(* IEC 61131-3 sources: Yaha/Documentation/Infomaterial/OSCAT/pcworx_basic_333/module_export (part 2) *)

(* ---- CALIBRATE.ST ---- *)
(*@PROPERTIES_EX@
TYPE: POU
LOCALE: 0
IEC_LANGUAGE: ST
PLC_TYPE: independent
PROC_TYPE: independent
GROUP: ENGINEERING.MEASUREMENTS
*)
(*@KEY@:DESCRIPTION*)
version 1.3	11. mar. 2009
programmer 	hugo
tested BY	hans

Calibrate allows for offset and scale calibration of an analog input.
offset is calibrated to a stored reference Y_offset while CO is true.
after the offset is calibrated, scale can be calibrated to a reference value Y_scale while CS is true.
*)
(*@KEY@:END_DESCRIPTION*)
FUNCTION_BLOCK CALIBRATE

(*Group:Default*)

VAR_INPUT
	X :	REAL;
	CO :	BOOL;
	CS :	BOOL;
	Y_OFFSET :	REAL;
	Y_SCALE :	REAL;
END_VAR

VAR_OUTPUT
	Y :	REAL;
END_VAR

VAR RETAIN
	offset :	REAL;
	Scale :	REAL := 1.0;
END_VAR

(*@KEY@: WORKSHEET
NAME: CALIBRATE
IEC_LANGUAGE: ST
*)
(* check for calibration *)
IF CO THEN
	OFFSET := Y_Offset - X;
ELSIF CS THEN
	SCALE := Y_scale / (X + OFFSET);
END_IF;
(* calculate output *)
Y := (X + OFFSET) * SCALE;

(* revision history
hm 22.2.2007		rev 1.2
	changed VAR RETAIN PERSISTENT to VAR RETAIN for better compatibility
	wago lon contollers do not support persisitent

hm	11. mar. 2009	rev 1.3
	changed real constants to use dot syntax

*)
(*@KEY@: END_WORKSHEET *)
END_FUNCTION_BLOCK

(* ---- CAPITALIZE.ST ---- *)
(*@PROPERTIES_EX@
TYPE: POU
LOCALE: 0
IEC_LANGUAGE: ST
PLC_TYPE: independent
PROC_TYPE: independent
GROUP: STRINGS
*)
(*@KEY@:DESCRIPTION*)
version 1.1	29. mar 2008
programmer 	hugo
tested by	tobias

uppercase returns str while all letters a..z and ä,ö,ü are converted to uppercase
(*@KEY@:END_DESCRIPTION*)
FUNCTION_BLOCK CAPITALIZE

(*Group:Default*)

VAR_INPUT
	STR :	STRING;
END_VAR

VAR_OUTPUT
	CAPITALIZE :	STRING;
END_VAR

VAR
	char :	BYTE;
	char2 :	BYTE;
	pos :	INT;
	L :	INT;
	first :	BOOL;
	str_temp :	STRING;
END_VAR

(*@KEY@: WORKSHEET
NAME: CAPITALIZE
IEC_LANGUAGE: ST
*)
CAPITALIZE := str;
first := TRUE;
L := LEN(str);
FOR pos := 1 TO L DO
   	char := INT_TO_BYTE(GET_CHAR(str,pos));
	IF first THEN
		char2 := TO_UPPER(char);
    	IF char <> char2 THEN
    		str_temp := CAPITALIZE;
      		CAPITALIZE := REPLACE(str_temp,BYTE_TO_STRING(char2,'%c'),1,pos);
		END_IF;
	END_IF;
	(* remember in first if the next char needs to capitalized *)
	first := char = BYTE#32;
END_FOR;

(* revision histroy
hm		4. mar 2008	rev 1.0
	original release

hm	29. mar. 2008	rev 1.1
	changed STRING to STRING(STRING_LENGTH)
*)
(*@KEY@: END_WORKSHEET *)
END_FUNCTION_BLOCK

(* ---- CARG.ST ---- *)
(*@PROPERTIES_EX@
TYPE: POU
LOCALE: 0
IEC_LANGUAGE: ST
PLC_TYPE: independent
PROC_TYPE: independent
GROUP: MATHEMATICAL.COMPLEX
*)
(*@KEY@:DESCRIPTION*)
version 1.1	20. apr. 2008
programmer 	hugo
tested by	oscat

this function calculates the phase angle (argument) of a complex number
(*@KEY@:END_DESCRIPTION*)
FUNCTION_BLOCK CARG

(*Group:Default*)

VAR_INPUT
	X :	oscat_complex;
END_VAR

VAR_OUTPUT
	CARG :	REAL;
END_VAR

(*@KEY@: WORKSHEET
NAME: CARG
IEC_LANGUAGE: ST
*)
CARG := ATAN2(X.im, X.re);

(* revision history
hm	21. feb. 2008	rev 1.0
	original version

hm	20. apr. 2008	rev 1.1
	use ATAN2 instead of ATAN
*)
(*@KEY@: END_WORKSHEET *)
END_FUNCTION_BLOCK

(* ---- CASIN.ST ---- *)
(*@PROPERTIES_EX@
TYPE: POU
LOCALE: 0
IEC_LANGUAGE: ST
PLC_TYPE: independent
PROC_TYPE: independent
GROUP: MATHEMATICAL.COMPLEX
*)
(*@KEY@:DESCRIPTION*)
version 1.0	21 feb 2008
programmer 	hugo
tested by	oscat

this function calculates the arcus sinus function of a complex number
(*@KEY@:END_DESCRIPTION*)
FUNCTION_BLOCK CASIN

(*Group:Default*)

VAR_INPUT
	X :	oscat_complex;
END_VAR

VAR_OUTPUT
	CASIN :	oscat_complex;
END_VAR

VAR
	Y :	oscat_complex;
	CASINH :	CASINH;
END_VAR

(*@KEY@: WORKSHEET
NAME: CASIN
IEC_LANGUAGE: ST
*)
y.re := -x.im;
y.im := x.re;
CASINH(X:=y);
y := CASINH.CASINH;
CASIN.re := y.im;
CASIN.im := -y.re;

(* revision history
hm	21. feb 2008	rev 1.0
	original version

*)
(*@KEY@: END_WORKSHEET *)
END_FUNCTION_BLOCK

(* ---- CASINH.ST ---- *)
(*@PROPERTIES_EX@
TYPE: POU
LOCALE: 0
IEC_LANGUAGE: ST
PLC_TYPE: independent
PROC_TYPE: independent
GROUP: MATHEMATICAL.COMPLEX
*)
(*@KEY@:DESCRIPTION*)
version 1.0	21 feb 2008
programmer 	hugo
tested by	oscat

this function calculates the hyperbolic arcus sinus function of a complex number
(*@KEY@:END_DESCRIPTION*)
FUNCTION_BLOCK CASINH

(*Group:Default*)

VAR_INPUT
	X :	oscat_complex;
END_VAR

VAR_OUTPUT
	CASINH :	oscat_complex;
END_VAR

VAR
	Y :	oscat_complex;
	CLOG :	CLOG;
	CSQRT :	CSQRT;
END_VAR

(*@KEY@: WORKSHEET
NAME: CASINH
IEC_LANGUAGE: ST
*)
y.re := (X.re - X.im)*(X.re + X.im) + 1.0;
y.im := 2.0 * X.re * X.im;
CSQRT(X:=y);
y    := CSQRT.CSQRT;
y.re := y.re + x.re;
y.im := y.im + x.im;
CLOG(X:=y);
CASINH  := CLOG.CLOG;

(* revision history
hm	21. feb 2008	rev 1.0
	original version

*)
(*@KEY@: END_WORKSHEET *)
END_FUNCTION_BLOCK

(* ---- CATAN.ST ---- *)
(*@PROPERTIES_EX@
TYPE: POU
LOCALE: 0
IEC_LANGUAGE: ST
PLC_TYPE: independent
PROC_TYPE: independent
GROUP: MATHEMATICAL.COMPLEX
*)
(*@KEY@:DESCRIPTION*)
version 1.0	21 feb 2008
programmer 	hugo
tested by	oscat

this function calculates the complex arcus tangens
(*@KEY@:END_DESCRIPTION*)
FUNCTION_BLOCK CATAN

(*Group:Default*)

VAR_INPUT
	X :	oscat_complex;
END_VAR

VAR_OUTPUT
	CATAN :	oscat_complex;
END_VAR

VAR
	r2 :	REAL;
	num :	REAL;
	den :	REAL;
END_VAR

(*@KEY@: WORKSHEET
NAME: CATAN
IEC_LANGUAGE: ST
*)
r2 := x.re * x.re;
den := 1.0 - r2 - x.im * x.im;
CATAN.re := 0.5 * ATAN(2.0 * x.re / den);
num := x.im + 1.0;
num := r2 + num * num;
den := x.im - 1.0;
den := r2 + den * den;
CATAN.im := 0.25 * (LN(num)-LN(den));

(* revision history
hm	21. feb 2008	rev 1.0
	original version
*)
(*@KEY@: END_WORKSHEET *)
END_FUNCTION_BLOCK

(* ---- CATANH.ST ---- *)
(*@PROPERTIES_EX@
TYPE: POU
LOCALE: 0
IEC_LANGUAGE: ST
PLC_TYPE: independent
PROC_TYPE: independent
GROUP: MATHEMATICAL.COMPLEX
*)
(*@KEY@:DESCRIPTION*)
version 1.0	21 feb 2008
programmer 	hugo
tested by	oscat

this function calculates the complex arcus hyperbolic tangens
(*@KEY@:END_DESCRIPTION*)
FUNCTION_BLOCK CATANH

(*Group:Default*)

VAR_INPUT
	X :	oscat_complex;
END_VAR

VAR_OUTPUT
	CATANH :	oscat_complex;
END_VAR

VAR
	i2 :	REAL;
	num :	REAL;
	den :	REAL;
END_VAR

(*@KEY@: WORKSHEET
NAME: CATANH
IEC_LANGUAGE: ST
*)
i2 := x.im * x.im;
num := 1.0 + x.re;
num := i2 + num * num;
den := 1.0 - x.re;
den := i2 + den * den;
CATANH.re := 0.25 * (LN(num) - LN(den));
den := 1.0 - x.re * x.re - i2;
CATANH.im := 0.5 * ATAN(2.0 * x.im / den);

(* revision history
hm	21. feb 2008	rev 1.0
	original version

*)
(*@KEY@: END_WORKSHEET *)
END_FUNCTION_BLOCK

(* ---- CCON.ST ---- *)
(*@PROPERTIES_EX@
TYPE: POU
LOCALE: 0
IEC_LANGUAGE: ST
PLC_TYPE: independent
PROC_TYPE: independent
GROUP: MATHEMATICAL.COMPLEX
*)
(*@KEY@:DESCRIPTION*)
version 1.0	21 feb 2008
programmer 	hugo
tested by	oscat

this function calcucates the conjugation of a complex number
(*@KEY@:END_DESCRIPTION*)
FUNCTION_BLOCK CCON

(*Group:Default*)

VAR_INPUT
	X :	oscat_complex;
END_VAR

VAR_OUTPUT
	CCON :	oscat_complex;
END_VAR

(*@KEY@: WORKSHEET
NAME: CCON
IEC_LANGUAGE: ST
*)
CCON.re := x.re;
CCON.im := -x.im;

(* revision history
hm	21. feb 2008	rev 1.0
	original version

*)
(*@KEY@: END_WORKSHEET *)
END_FUNCTION_BLOCK

(* ---- CCOS.ST ---- *)
(*@PROPERTIES_EX@
TYPE: POU
LOCALE: 0
IEC_LANGUAGE: ST
PLC_TYPE: independent
PROC_TYPE: independent
GROUP: MATHEMATICAL.COMPLEX
*)
(*@KEY@:DESCRIPTION*)
version 1.0	21 feb 2008
programmer 	hugo
tested by	oscat

this function calculates the cosinus function of a complex number
(*@KEY@:END_DESCRIPTION*)
FUNCTION_BLOCK CCOS

(*Group:Default*)

VAR_INPUT
	X :	oscat_complex;
END_VAR

VAR_OUTPUT
	CCOS :	oscat_complex;
END_VAR

VAR
	CSET :	CSET;
	CCOSH :	CCOSH;
END_VAR

(*@KEY@: WORKSHEET
NAME: CCOS
IEC_LANGUAGE: ST
*)
CSET(RE:= -X.im,IM:=X.re);
CCOSH(X:=CSET.CSET);
CCOS := CCOSH.CCOSH;

(* revision history
hm	21. feb 2008	rev 1.0
	original version

*)
(*@KEY@: END_WORKSHEET *)
END_FUNCTION_BLOCK

(* ---- CCOSH.ST ---- *)
(*@PROPERTIES_EX@
TYPE: POU
LOCALE: 0
IEC_LANGUAGE: ST
PLC_TYPE: independent
PROC_TYPE: independent
GROUP: MATHEMATICAL.COMPLEX
*)
(*@KEY@:DESCRIPTION*)
version 1.0	21 feb 2008
programmer 	hugo
tested by	oscat

this function calculates the arcus tangens function of a complex number
(*@KEY@:END_DESCRIPTION*)
FUNCTION_BLOCK CCOSH

(*Group:Default*)

VAR_INPUT
	X :	oscat_complex;
END_VAR

VAR_OUTPUT
	CCOSH :	oscat_complex;
END_VAR

(*@KEY@: WORKSHEET
NAME: CCOSH
IEC_LANGUAGE: ST
*)
CCOSH.re := cosH(x.re) * COS(x.im);
CCOSH.im := sinH(x.re) * SIN(x.im);

(* revision history
hm	21. feb 2008	rev 1.0
	original version

*)
(*@KEY@: END_WORKSHEET *)
END_FUNCTION_BLOCK

(* ---- CDIV.ST ---- *)
(*@PROPERTIES_EX@
TYPE: POU
LOCALE: 0
IEC_LANGUAGE: ST
PLC_TYPE: independent
PROC_TYPE: independent
GROUP: MATHEMATICAL.COMPLEX
*)
(*@KEY@:DESCRIPTION*)
version 1.0	21 feb 2008
programmer 	hugo
tested by	oscat

this function divides two complex numbers
(*@KEY@:END_DESCRIPTION*)
FUNCTION_BLOCK CDIV

(*Group:Default*)

VAR_INPUT
	X :	oscat_complex;
	Y :	oscat_complex;
END_VAR

VAR_OUTPUT
	CDIV :	oscat_complex;
END_VAR

VAR
	temp :	REAL;
END_VAR

(*@KEY@: WORKSHEET
NAME: CDIV
IEC_LANGUAGE: ST
*)
temp := Y.re * Y.re + Y.im * Y.im;
IF temp = 0.0 THEN CDIV.re := 0.0;CDIV.im := 0.0;RETURN;END_IF;
CDIV.re := (X.re * Y.re + X.im * Y.im) / temp;
CDIV.im := (X.im * Y.re - X.re * Y.im) / temp;

(* revision history
hm	21. feb 2008	rev 1.0
	original version

*)
(*@KEY@: END_WORKSHEET *)
END_FUNCTION_BLOCK

(* ---- CEXP.ST ---- *)
(*@PROPERTIES_EX@
TYPE: POU
LOCALE: 0
IEC_LANGUAGE: ST
PLC_TYPE: independent
PROC_TYPE: independent
GROUP: MATHEMATICAL.COMPLEX
*)
(*@KEY@:DESCRIPTION*)
version 1.0	21 feb 2008
programmer 	hugo
tested by	oscat

this function calculates the complex exponent
(*@KEY@:END_DESCRIPTION*)
FUNCTION_BLOCK CEXP

(*Group:Default*)

VAR_INPUT
	X :	oscat_complex;
END_VAR

VAR_OUTPUT
	CEXP :	oscat_complex;
END_VAR

VAR
	Temp :	REAL;
END_VAR

(*@KEY@: WORKSHEET
NAME: CEXP
IEC_LANGUAGE: ST
*)
temp := EXP(X.re);
CEXP.re := temp * COS(X.im);
CEXP.im := temp * SIN(X.im);

(* revision history
hm	21. feb 2008	rev 1.0
	original version

*)
(*@KEY@: END_WORKSHEET *)
END_FUNCTION_BLOCK

(* ---- CHARCODE.ST ---- *)
(*@PROPERTIES_EX@
TYPE: POU
LOCALE: 0
IEC_LANGUAGE: ST
PLC_TYPE: independent
PROC_TYPE: independent
GROUP: STRINGS
*)
(*@KEY@:DESCRIPTION*)
version 1.1		19. oct. 2008
programmer 		hugo
tested by		hugo

CHARCODE converts a HTML Character NAME INTO ITS code
'äuml' is convterted to ä
'euro' is converted to €
(*@KEY@:END_DESCRIPTION*)
FUNCTION_BLOCK CHARCODE

(*Group:IN_OUT*)

VAR_INPUT
	STR :	oscat_STRING10;
END_VAR

VAR_OUTPUT
	CHARCODE :	BYTE;
END_VAR

VAR
	found :	oscat_STRING1;
	search :	oscat_STRING10;
	pos :	INT;
	CODE :	CODE;
	i :	INT;
	SETUP_CHARNAMES :	SETUP_CHARNAMES;
	CHARNAMES :	oscat_CHARNAMES;
END_VAR

(*@KEY@: WORKSHEET
NAME: CHARCODE
IEC_LANGUAGE: ST
*)
SETUP_CHARNAMES(CHARNAMES:=CHARNAMES);
CHARNAMES:=SETUP_CHARNAMES.CHARNAMES;

IF LEN(str) = 1 THEN
    CODE(STR:=STR,POS:=1);
    CHARCODE:=CODE.CODE;
ELSIF LEN(str) > 0 THEN
	(* construct search string *)
	search := CONCAT('&', str);
	search := CONCAT(search, ';');
	WHILE pos = 0 AND (i < 11) DO
		i := i + 1;
		pos := FIND(CHARNAMES[i], search);
	END_WHILE;
	found := MID(CHARNAMES[i], 1, pos - 1);
    CODE(STR:=found,POS:=1);
    CHARCODE:=CODE.CODE;
END_IF;

(* revision history
hm	13. may. 2008	rev 1.0
	original version

hm	19. oct. 2008	rev 1.1
	changed setup constants

hm	24. oct. 2008	rev 1.2
	optimized code
*)
(*@KEY@: END_WORKSHEET *)
END_FUNCTION_BLOCK

(* ---- CHARNAME.ST ---- *)
(*@PROPERTIES_EX@
TYPE: POU
LOCALE: 0
IEC_LANGUAGE: ST
PLC_TYPE: independent
PROC_TYPE: independent
GROUP: STRINGS
*)
(*@KEY@:DESCRIPTION*)
version 1.4		17. dec. 2008
programmer 		hugo
tested by		oscat

CHARNAME converts a Character code into its HTML character name
ä is convterted to 'äuml'
€ is converted to 'euro'
the character itself is returned if no name is available for the character
(*@KEY@:END_DESCRIPTION*)
FUNCTION_BLOCK CHARNAME

(*Group:IN_OUT*)

VAR_INPUT
	C :	BYTE;
END_VAR

VAR_OUTPUT
	CHARNAME :	oscat_STRING10;
END_VAR

VAR
	CHARNAME2 :	oscat_STRING10;
	pos :	INT;
	i :	INT;
	CHR_TO_STRING :	CHR_TO_STRING;
	SETUP_CHARNAMES :	SETUP_CHARNAMES;
	CHARNAMES :	oscat_CHARNAMES;
END_VAR

(*@KEY@: WORKSHEET
NAME: CHARNAME
IEC_LANGUAGE: ST
*)
SETUP_CHARNAMES(CHARNAMES:=CHARNAMES);
CHARNAMES:=SETUP_CHARNAMES.CHARNAMES;

IF C <> BYTE#0 THEN
	(* construct search string from code followed by $ sign, also clear charname string*)
	CHR_TO_STRING(C:=C);
	CHARNAME := CHR_TO_STRING.CHR_TO_STRING;
	CHARNAME2 := CONCAT(CHARNAME,'&');
	CHARNAME := CONCAT(';', CHARNAME2);
	WHILE pos = 0 AND (i < 11) DO
		i := i + 1;
		pos := FIND(CHARNAMES[i], CHARNAME);
	END_WHILE;
	IF pos > 0 THEN
		CHARNAME := MID(CHARNAMES[i], 10, pos + 3);
		(* search for end of name and truncate *)
		pos := FIND(CHARNAME, ';');
		CHARNAME := LEFT(CHARNAME,pos - 1);
	ELSE
		CHR_TO_STRING(C:=C);
		CHARNAME := CHR_TO_STRING.CHR_TO_STRING;
	END_IF;
ELSE
	CHARNAME := '';
END_IF;

(* revision history
hm	13. may. 2008	rev 1.0
	original version

hm	16. jun. 2008	rev 1.1
	changed nested call of concat for better compatibility

hm	19. oct. 2008	rev 1.2
	changes setup constants

hm	24. oct. 2008	rev 1.3
	new code for high performance

hm	17. dec. 2008	rev 1.4
	changed function chr to chr_to_string
*)
(*@KEY@: END_WORKSHEET *)
END_FUNCTION_BLOCK

(* ---- CHK_REAL.ST ---- *)
(*@PROPERTIES_EX@
TYPE: POU
LOCALE: 0
IEC_LANGUAGE: ST
PLC_TYPE: independent
PROC_TYPE: independent
GROUP: LOGIC.GATE_LOGIC
*)
(*@KEY@:DESCRIPTION*)
version 1.0	20. jan. 2011
programmer 	hugo
tested by	tobias

this function checks a floating point variable of type real (IEEE754-32Bits) for NAN and infinity
RETURN values: #0 = normal value, #20 = +infinity, #40 = -infinty, #80 = NAN

(*@KEY@:END_DESCRIPTION*)
FUNCTION_BLOCK CHK_REAL

(*Group:Default*)

VAR_INPUT
	X :	REAL;
END_VAR

VAR_OUTPUT
	CHK_REAL :	BYTE;
END_VAR

VAR
	tmp :	DWORD;
	REAL_TO_DW :	REAL_TO_DW;
END_VAR

(*@KEY@: WORKSHEET
NAME: CHK_REAL
IEC_LANGUAGE: ST
*)
REAL_TO_DW(X:=X); (* move real to dword, real_to_dword does not work becasze it treats dword as a number on many systems *)
tmp := ROL(REAL_TO_DW.REAL_TO_DW,1);(* rotate left foir easy checking, sign will be at lease significant digit *)
IF tmp < DWORD#16#FF000000 THEN
	CHK_REAL := BYTE#16#00;	(* normalized and denormalized numbers *)
ELSIF tmp = DWORD#16#FF000000 THEN
	CHK_REAL := BYTE#16#20;	(* X is +infinity see IEEE754 *)
ELSIF tmp = DWORD#16#FF000001 THEN
	CHK_REAL := BYTE#16#40;	(* X is -infinity see IEEE754 *)
ELSE
	CHK_REAL := BYTE#16#80;	(* X is NAN see IEEE754 *)
END_IF;

(* revision history
hm	 20. jan. 2011	rev 1.0
	original version

*)

(*@KEY@: END_WORKSHEET *)
END_FUNCTION_BLOCK

(* ---- CHR_TO_STRING.ST ---- *)
(*@PROPERTIES_EX@
TYPE: POU
LOCALE: 0
IEC_LANGUAGE: ST
PLC_TYPE: independent
PROC_TYPE: independent
GROUP: STRINGS
*)
(*@KEY@:DESCRIPTION*)
version 1.3	17. dec. 2008
programmer 	hugo
tested by	oscat

CHR creates a character from a byte input and stuffs it in a one character length string.
(*@KEY@:END_DESCRIPTION*)
FUNCTION_BLOCK CHR_TO_STRING

(*Group:x*)

VAR_INPUT
	C :	BYTE;
END_VAR

VAR_OUTPUT
	CHR_TO_STRING :	oscat_STRING1;
END_VAR

(*@KEY@: WORKSHEET
NAME: CHR_TO_STRING
IEC_LANGUAGE: ST
*)
CHR_TO_STRING := BYTE_TO_STRING(C,'%c');

(* revision history
hm	16 jan 2007		rev 1.0
	original version

hm	4. feb. 2008	rev 1.1
	return string would not be terminated properly

hm	29. mar. 2008	rev 1.2
	changed STRING to STRING(1)

hm	17. dec. 2008	rev 1.3
	changed name of function from chr to chr_to_string
*)
(*@KEY@: END_WORKSHEET *)
END_FUNCTION_BLOCK

(* ---- CINV.ST ---- *)
(*@PROPERTIES_EX@
TYPE: POU
LOCALE: 0
IEC_LANGUAGE: ST
PLC_TYPE: independent
PROC_TYPE: independent
GROUP: MATHEMATICAL.COMPLEX
*)
(*@KEY@:DESCRIPTION*)
version 1.0	21 feb 2008
programmer 	hugo
tested by	oscat

this function calculates the inverse of a complex numbers (1 / X)
(*@KEY@:END_DESCRIPTION*)
FUNCTION_BLOCK CINV

(*Group:Default*)

VAR_INPUT
	X :	oscat_complex;
END_VAR

VAR_OUTPUT
	CINV :	oscat_complex;
END_VAR

VAR
	temp :	REAL;
END_VAR

(*@KEY@: WORKSHEET
NAME: CINV
IEC_LANGUAGE: ST
*)
temp := X.re * X.re + X.im * X.im;
IF temp = 0.0 THEN CINV.re := 0.0;CINV.im := 0.0;RETURN;END_IF;
CINV.re := X.re / temp;
CINV.im := -X.im / temp;

(* revision history
hm	21. feb 2008	rev 1.0
	original version

*)
(*@KEY@: END_WORKSHEET *)
END_FUNCTION_BLOCK

(* ---- CLEAN.ST ---- *)
(*@PROPERTIES_EX@
TYPE: POU
LOCALE: 0
IEC_LANGUAGE: ST
PLC_TYPE: independent
PROC_TYPE: independent
GROUP: STRINGS
*)
(*@KEY@:DESCRIPTION*)
version 1.0	18. jun. 2008
programmer 	hugo
tested by	oscat

Clean deletes all characters from a string except the ones specified in CX.
(*@KEY@:END_DESCRIPTION*)
FUNCTION_BLOCK CLEAN

(*Group:lokal*)

(*Group:IN_OUT*)

VAR_INPUT
	IN :	oscat_STRING250;
	CX :	STRING;
END_VAR

VAR_OUTPUT
	CLEAN :	oscat_STRING250;
END_VAR

VAR
	pos :	INT;
	stop :	INT;
	char :	oscat_STRING1;
END_VAR

(*@KEY@: WORKSHEET
NAME: CLEAN
IEC_LANGUAGE: ST
*)
(* copy input string *)
CLEAN := IN;
stop := LEN(in);
pos := 1;
WHILE pos <= stop DO
    char := MID(CLEAN, 1, pos);
	IF FIND(cx,char) > 0 THEN
		(* charcter found skip to next one *)
		pos := pos + 1;
	ELSE
		(* wrong chracter needs to be deleted *)
		CLEAN := DELETE(CLEAN, 1, pos);
		stop := stop - 1;	(* the string is one character shorter now *)
	END_IF;
END_WHILE;

(* revision history

hm		18. jun. 2008	rev 1.0
	original version

*)
(*@KEY@: END_WORKSHEET *)
END_FUNCTION_BLOCK

(* ---- CLICK_CNT.ST ---- *)
(*@PROPERTIES_EX@
TYPE: POU
LOCALE: 0
IEC_LANGUAGE: ST
PLC_TYPE: independent
PROC_TYPE: independent
GROUP: LOGIC.GENERATORS
*)
(*@KEY@:DESCRIPTION*)
version 1.0	16. jul. 2008
programmer 	hugo
tested by	oscat

this Module decodes a specified number of clicks.
the output trig is high for one cycle if N clicks are present within a specified time TC.
(*@KEY@:END_DESCRIPTION*)
FUNCTION_BLOCK CLICK_CNT

(*Group:Default*)

VAR_INPUT
	IN :	BOOL;
	N :	INT;
	TC :	TIME;
END_VAR

VAR_OUTPUT
	Q :	BOOL;
END_VAR

VAR
	tx :	TP;
	edge :	BOOL;
	cnt :	INT := INT#-1;
END_VAR

(*@KEY@: WORKSHEET
NAME: CLICK_CNT
IEC_LANGUAGE: ST
*)
(* Q shall only be active for one cycle only *)
Q := FALSE;

IF in AND NOT edge AND NOT tx.q THEN
	(* a rising edge on in sets the counter to 0 *)
	cnt := 0;
ELSIF tx.Q AND NOT IN AND edge THEN
	(* count falling edges when tp.q is true *)
	cnt := cnt + 1;
ELSIF NOT tx.Q THEN
	Q := cnt=N;
	cnt := -1;
END_IF;

(* remember the status of IN *)
edge := IN;
tx(in := IN, pt := TC);

(* revision history

hm 	16. jul. 2008	rev 1.0
	original version released

*)
(*@KEY@: END_WORKSHEET *)
END_FUNCTION_BLOCK

(* ---- CLICK_DEC.ST ---- *)
(*@PROPERTIES_EX@
TYPE: POU
LOCALE: 0
IEC_LANGUAGE: ST
PLC_TYPE: independent
PROC_TYPE: independent
GROUP: LOGIC.GENERATORS
*)
(*@KEY@:DESCRIPTION*)
version 1.1	14. mar. 2009
programmer 	hugo
tested by	oscat

this Module detects a rising edge on In and decodes the amount of falling edges (Pulses) within a specified time TC.
the outputs Q0..Q3 will go true for one cycle and the amount of clicks within a specified time TC.
if only a rising egde is detected within TC Q0 will respond, Q1 for 1 pulse and so on..

(*@KEY@:END_DESCRIPTION*)
FUNCTION_BLOCK CLICK_DEC

(*Group:Default*)

VAR_INPUT
	IN :	BOOL;
	TC :	TIME;
END_VAR

VAR_OUTPUT
	Q0 :	BOOL;
	Q1 :	BOOL;
	Q2 :	BOOL;
	Q3 :	BOOL;
END_VAR

VAR
	tx :	TP;
	edge :	BOOL;
	cnt :	INT := INT#-1;
END_VAR

(*@KEY@: WORKSHEET
NAME: CLICK_DEC
IEC_LANGUAGE: ST
*)
(* Q shall only be active for one cycle only *)
IF in = FALSE THEN
	Q0 := FALSE;
	Q1 := FALSE;
	Q2 := FALSE;
	Q3 := FALSE;
END_IF;

IF in AND NOT edge AND NOT tx.q THEN
	(* a rising edge on in sets the counter to 0 *)
	cnt := 0;
ELSIF tx.Q AND NOT IN AND edge THEN
	(* count falling edges when tp.q is true *)
	cnt := cnt + 1;
ELSIF NOT tx.Q THEN
	CASE cnt OF
		0 : Q0 := TRUE;
		1 : Q1 := TRUE;
		2 : Q2 := TRUE;
		3 : Q3 := TRUE;
	END_CASE;
	cnt := -1;
END_IF;

(* remember the status of IN *)
edge := IN;
tx(in := IN, pt := TC);

(* revision history

hm 17. jul. 2008	rev 1.0
	original version released

hm	14. mar. 2009	rev 1.1
	removed double assignments

*)
(*@KEY@: END_WORKSHEET *)
END_FUNCTION_BLOCK

(* ---- CLK_DIV.ST ---- *)
(*@PROPERTIES_EX@
TYPE: POU
LOCALE: 0
IEC_LANGUAGE: ST
PLC_TYPE: independent
PROC_TYPE: independent
GROUP: LOGIC.GENERATORS
*)
(*@KEY@:DESCRIPTION*)
version 1.1	2 jan 2008
programmer 	hugo
tested by	tobias

this is a clock divider
each output divides the signal by 2
Q0 = clk / 2 , Q1 = Q0 / 2 and so on.
the outputs have a 50% duty cycle each.
(*@KEY@:END_DESCRIPTION*)
FUNCTION_BLOCK CLK_DIV

(*Group:Default*)

VAR_INPUT
	CLK :	BOOL;
	RST :	BOOL;
END_VAR

VAR_OUTPUT
	Q0 :	BOOL := FALSE;
	Q1 :	BOOL := FALSE;
	Q2 :	BOOL := FALSE;
	Q3 :	BOOL := FALSE;
	Q4 :	BOOL := FALSE;
	Q5 :	BOOL := FALSE;
	Q6 :	BOOL := FALSE;
	Q7 :	BOOL := FALSE;
END_VAR

VAR
	cnt :	BYTE := 0;
END_VAR

(*@KEY@: WORKSHEET
NAME: CLK_DIV
IEC_LANGUAGE: ST
*)
IF rst THEN
	cnt:= BYTE#0;
	Q0 := FALSE;
	Q1 := FALSE;
	Q2 := FALSE;
	Q3 := FALSE;
	Q4 := FALSE;
	Q5 := FALSE;
	Q6 := FALSE;
	Q7 := FALSE;
ELSIF clk THEN
	cnt:= USINT_TO_BYTE(BYTE_TO_USINT(cnt) + USINT#1);

    Q0 := BIT_OF_DWORD(BYTE_TO_DWORD(cnt),0); (* Q0 := cnt.X0; *)
    Q1 := BIT_OF_DWORD(BYTE_TO_DWORD(cnt),1); (* Q1 := cnt.X1; *)
    Q2 := BIT_OF_DWORD(BYTE_TO_DWORD(cnt),2); (* Q2 := cnt.X2; *)
    Q3 := BIT_OF_DWORD(BYTE_TO_DWORD(cnt),3); (* Q3 := cnt.X3; *)
    Q4 := BIT_OF_DWORD(BYTE_TO_DWORD(cnt),4); (* Q4 := cnt.X4; *)
    Q5 := BIT_OF_DWORD(BYTE_TO_DWORD(cnt),5); (* Q5 := cnt.X5; *)
    Q6 := BIT_OF_DWORD(BYTE_TO_DWORD(cnt),6); (* Q6 := cnt.X6; *)
    Q7 := BIT_OF_DWORD(BYTE_TO_DWORD(cnt),7); (* Q7 := cnt.X7; *)

END_IF;

(* revision history
hm	4. aug. 2006	rev 1.0
	original version

hm	2. jan 2008		rev 1.1
	improved performance

*)
(*@KEY@: END_WORKSHEET *)
END_FUNCTION_BLOCK

(* ---- CLK_N.ST ---- *)
(*@PROPERTIES_EX@
TYPE: POU
LOCALE: 0
IEC_LANGUAGE: ST
PLC_TYPE: independent
PROC_TYPE: independent
GROUP: LOGIC.GENERATORS
*)
(*@KEY@:DESCRIPTION*)
version 1.0	17 sep 2007
programmer 	hugo
tested by	tobias

clk_N uses the internal sps time to generate one pulse every N ms
every pulse is only valid for one cycle so that a edge trigger is not necessary
clk_gen generates pulses depending on the accuracy of the system clock.
The input N controlls the period time of the clock.
N=0 equals 2ms, N=1 equals 4ms, N=2 equals 8ms, N=3 equals 16ms ....

be careful, 1ms clocks will only work on very powerful sps cpu's
(*@KEY@:END_DESCRIPTION*)
FUNCTION_BLOCK CLK_N

(*Group:Default*)

VAR_INPUT
	N :	INT;
END_VAR

VAR_OUTPUT
	Q :	BOOL;
END_VAR

VAR
	T_PLC_MS :	T_PLC_MS;
	edge :	BOOL;
	clk :	BOOL;
END_VAR

(*@KEY@: WORKSHEET
NAME: CLK_N
IEC_LANGUAGE: ST
*)
T_PLC_MS();
clk := BIT_OF_DWORD(SHR(UDINT_TO_DWORD(T_PLC_MS.T_PLC_MS),N),0);
Q := clk XOR edge;
edge := clk;

(* revision history
hm	16. dec 2007		rev 1.0
	original version

*)
(*@KEY@: END_WORKSHEET *)
END_FUNCTION_BLOCK

(* ---- CLK_PRG.ST ---- *)
(*@PROPERTIES_EX@
TYPE: POU
LOCALE: 0
IEC_LANGUAGE: ST
PLC_TYPE: independent
PROC_TYPE: independent
GROUP: LOGIC.GENERATORS
*)
(*@KEY@:DESCRIPTION*)
version 1.3	25. oct. 2008
programmer 	hugo
tested by	tobias

clk_prg uses the internal sps time to generate a clock with programmable period time.
the period time is defined for 10ms .. 65s
the first cycle after start is a clk pulse and then depending on the programmed period time a delay.
every pulse is only valid for one cycle.
the accuracy of clk_prg is depending on the accuracy of the system clock.
(*@KEY@:END_DESCRIPTION*)
FUNCTION_BLOCK CLK_PRG

(*Group:Default*)

VAR_INPUT
	PT :	TIME := T#10ms;
END_VAR

VAR_OUTPUT
	Q :	BOOL;
END_VAR

VAR
	init :	BOOL := FALSE;
	last :	TIME;
	tx :	TIME;
	T_PLC_MS :	T_PLC_MS;
END_VAR

(*@KEY@: WORKSHEET
NAME: CLK_PRG
IEC_LANGUAGE: ST
*)
(* read system time *)
T_PLC_MS();
tx:= UDINT_TO_TIME(T_PLC_MS.T_PLC_MS);

(* initialize on startup *)
IF NOT init THEN
	init := TRUE;
	last := tx - pt;
END_IF;

(* generate output pulse when next_pulse is reached *)
Q := tx - last >= pt;
IF Q THEN last := tx; END_IF;

(* revision hiostory

hm 25 feb 2007	rev 1.1
	rewritten code for higher performance
	pt can now be changed during runtime

hm	17. sep 2007	rev 1.2
	replaced time() with t_plc_ms() for compatibility reasons

hm	25. oct. 2008	rev 1.3
	optimized code

*)
(*@KEY@: END_WORKSHEET *)
END_FUNCTION_BLOCK

(* ---- CLK_PULSE.ST ---- *)
(*@PROPERTIES_EX@
TYPE: POU
LOCALE: 0
IEC_LANGUAGE: ST
PLC_TYPE: independent
PROC_TYPE: independent
GROUP: LOGIC.GENERATORS
*)
(*@KEY@:DESCRIPTION*)
version 1.2		16 feb 2011
programmer 	    hugo
tested by		oscat

clk_pulse uses the internal sps time to generate a clock with programmable period time.
the period time is defined for 10ms .. 65s.
pulse generation is continuous if N = 0 and for n pulses otherwise.
the first cycle after start is a clk pulse and then depending on the programmed period time a delay.
every pulse is only valid for one cycle so that a edge trigger is not necessary
clk_prg depending on the accuracy of the system clock.

(*@KEY@:END_DESCRIPTION*)
FUNCTION_BLOCK CLK_PULSE

(*Group:Default*)

VAR_INPUT
	PT :	TIME;
	N :	INT;
	RST :	BOOL;
END_VAR

VAR_OUTPUT
	Q :	BOOL;
	CNT :	INT;
	RUN :	BOOL;
END_VAR

VAR
	tx :	UDINT;
	tn :	UDINT;
	init :	BOOL;
	T_PLC_MS :	T_PLC_MS;
END_VAR

(*@KEY@: WORKSHEET
NAME: CLK_PULSE
IEC_LANGUAGE: ST
*)
(* read system *)
T_PLC_MS();
tx:= T_PLC_MS.T_PLC_MS;
Q := FALSE;				(* reset Q we generate pulses only for one cycle *)
RUN := CNT < N;

IF NOT init OR RST THEN
	init := TRUE;
	CNT := 0;
	tn := tx - TIME_TO_UDINT(PT);
	RUN := FALSE;
ELSIF (cnt < N OR N = 0) AND tx - tn >= TIME_TO_UDINT(PT) THEN		(* generate a pulse *)
	CNT := CNT + 1;
	Q := TRUE;
	tn := tn + TIME_TO_UDINT(PT);
END_IF;

(* revision history
hm		4. aug 2006		rev 1.0
	original version

hm		17. sep 2007	rev 1.1
	replaced time() with T_PLC_S() for compatblity reasons

hm		16. feb. 2011	rev 1.2
	fixed an error when timer overflows
*)
(*@KEY@: END_WORKSHEET *)
END_FUNCTION_BLOCK

(* ---- CLOG.ST ---- *)
(*@PROPERTIES_EX@
TYPE: POU
LOCALE: 0
IEC_LANGUAGE: ST
PLC_TYPE: independent
PROC_TYPE: independent
GROUP: MATHEMATICAL.COMPLEX
*)
(*@KEY@:DESCRIPTION*)
version 1.1	20. apr. 2008
programmer 	hugo
tested by	oscat

this function calculates the complex natural (base e) logarithm
(*@KEY@:END_DESCRIPTION*)
FUNCTION_BLOCK CLOG

(*Group:Default*)

VAR_INPUT
	X :	oscat_complex;
END_VAR

VAR_OUTPUT
	CLOG :	oscat_complex;
END_VAR

(*@KEY@: WORKSHEET
NAME: CLOG
IEC_LANGUAGE: ST
*)
CLOG.re := LN(HYPOT(X.re, X.im));
CLOG.im := ATAN2(X.im, X.re);

(* revision history
hm	21. feb 2008	rev 1.0
	original version

hm	20. apr. 2008	rev 1.1
	use ATAN2 instead of ATAN
*)
(*@KEY@: END_WORKSHEET *)
END_FUNCTION_BLOCK

(* ---- CMUL.ST ---- *)
(*@PROPERTIES_EX@
TYPE: POU
LOCALE: 0
IEC_LANGUAGE: ST
PLC_TYPE: independent
PROC_TYPE: independent
GROUP: MATHEMATICAL.COMPLEX
*)
(*@KEY@:DESCRIPTION*)
version 1.0	21 feb 2008
programmer 	hugo
tested by	oscat

this function multiplies two complex numbers
(*@KEY@:END_DESCRIPTION*)
FUNCTION_BLOCK CMUL

(*Group:Default*)

VAR_INPUT
	X :	oscat_complex;
	Y :	oscat_complex;
END_VAR

VAR_OUTPUT
	CMUL :	oscat_complex;
END_VAR

(*@KEY@: WORKSHEET
NAME: CMUL
IEC_LANGUAGE: ST
*)
CMUL.re := X.re * Y.re - X.im * Y.im;
CMUL.im := X.re * Y.im + X.im * Y.re;

(* revision history
hm	21. feb 2008	rev 1.0
	original version

*)
(*@KEY@: END_WORKSHEET *)
END_FUNCTION_BLOCK

(* ---- CODE.ST ---- *)
(*@PROPERTIES_EX@
TYPE: POU
LOCALE: 0
IEC_LANGUAGE: ST
PLC_TYPE: independent
PROC_TYPE: independent
GROUP: STRINGS
*)
(*@KEY@:DESCRIPTION*)
version 1.1	29. mar. 2008
programmer 	hugo
tested by	tobias

code extracts the code of a character at position POS of a string STR.
(*@KEY@:END_DESCRIPTION*)
FUNCTION_BLOCK CODE

(*Group:Default*)

VAR_INPUT
	STR :	STRING;
	POS :	INT;
END_VAR

VAR_OUTPUT
	CODE :	BYTE;
END_VAR

(*@KEY@: WORKSHEET
NAME: CODE
IEC_LANGUAGE: ST
*)
IF pos < 1 OR pos > LEN(str) THEN
	CODE := BYTE#0;
	RETURN;
ELSE
    CODE := INT_TO_BYTE(GET_CHAR(STR,POS));
END_IF;

(* revision history
hm	9. mar. 2008	rev 1.0
	original version

hm	29. mar. 2008	rev 1.1
	changed STRING to STRING(STRING_LENGTH)
*)
(*@KEY@: END_WORKSHEET *)
END_FUNCTION_BLOCK

(* ---- CODE_250.ST ---- *)
(*@PROPERTIES_EX@
TYPE: POU
LOCALE: 0
IEC_LANGUAGE: ST
PLC_TYPE: independent
PROC_TYPE: independent
GROUP: STRINGS
*)
(*@KEY@:DESCRIPTION*)

(*@KEY@:END_DESCRIPTION*)
FUNCTION_BLOCK CODE_250

(*Group:Default*)

VAR_INPUT
	STR :	oscat_STRING250;
	POS :	INT;
END_VAR

VAR_OUTPUT
	CODE :	BYTE;
END_VAR

(*@KEY@: WORKSHEET
NAME: CODE_250
IEC_LANGUAGE: ST
*)
IF pos < 1 OR pos > LEN(str) THEN
	CODE := BYTE#0;
	RETURN;
ELSE
    CODE := INT_TO_BYTE(GET_CHAR(STR,POS));
END_IF;

(* revision history
hm	9. mar. 2008	rev 1.0
	original version

hm	29. mar. 2008	rev 1.1
	changed STRING to STRING(STRING_LENGTH)
*)
(*@KEY@: END_WORKSHEET *)
END_FUNCTION_BLOCK

(* ---- CONTROL_SET1.ST ---- *)
(*@PROPERTIES_EX@
TYPE: POU
LOCALE: 0
IEC_LANGUAGE: ST
PLC_TYPE: independent
PROC_TYPE: independent
GROUP: ENGINEERING.CONTROL
*)
(*@KEY@:DESCRIPTION*)
version 1.1	11. mar. 2009
programmer 	hugo
tested by	tobias

takahashi calculates controller parameters for P, PI and PID controllers based on the ziegler nichols method.

(*@KEY@:END_DESCRIPTION*)
FUNCTION_BLOCK CONTROL_SET1

(*Group:Default*)

VAR_INPUT
	KT :	REAL;
	TT :	REAL;
	PI :	BOOL;
	PID :	BOOL;
	P_K :	REAL := 0.5;
	PI_K :	REAL := 0.45;
	PI_TN :	REAL := 0.83;
	PID_K :	REAL := 0.6;
	PID_TN :	REAL := 0.5;
	PID_TV :	REAL := 0.125;
END_VAR

VAR_OUTPUT
	KP :	REAL;
	TN :	REAL;
	TV :	REAL;
	KI :	REAL;
	KD :	REAL;
END_VAR

(*@KEY@: WORKSHEET
NAME: CONTROL_SET1
IEC_LANGUAGE: ST
*)
IF pi AND PID THEN
	KP := 0.0;
	TN := 0.0;
	TV := 0.0;
ELSIF PID THEN
	KP := PID_K * Kt;
	TN := PID_TN * Tt;
	TV := PID_TV * Tt;
ELSIF PI THEN
	KP := PI_K * Kt;
	TN := PI_TN * Tt;
ELSE
	KP := P_K * Kt;
END_IF;

(* KI and KD are calculated *)
IF tn > 0.0 THEN KI := KP / TN; ELSE KI := 0.0; END_IF;
KD := KP * TV;

(* revision history
hm	4. nov 2007	rev 1.0
	original version

hm	11. mar. 2009	rev 1.1
	real constants updated to new systax using dot

*)
(*@KEY@: END_WORKSHEET *)
END_FUNCTION_BLOCK

(* ---- CONTROL_SET2.ST ---- *)
(*@PROPERTIES_EX@
TYPE: POU
LOCALE: 0
IEC_LANGUAGE: ST
PLC_TYPE: independent
PROC_TYPE: independent
GROUP: ENGINEERING.CONTROL
*)
(*@KEY@:DESCRIPTION*)
version 1.1	11. mar. 2009
programmer 	hugo
tested by	tobias

takahashi calculates controller parameters for P, PI and PID controllers based on the ziegler nichols method.

(*@KEY@:END_DESCRIPTION*)
FUNCTION_BLOCK CONTROL_SET2

(*Group:Default*)

VAR_INPUT
	KS :	REAL;
	TU :	REAL;
	TG :	REAL;
	PI :	BOOL;
	PID :	BOOL;
	P_K :	REAL := 1.0;
	PI_K :	REAL := 0.9;
	PI_TN :	REAL := 3.33;
	PID_K :	REAL := 1.2;
	PID_TN :	REAL := 2.0;
	PID_TV :	REAL := 0.5;
END_VAR

VAR_OUTPUT
	KP :	REAL;
	TN :	REAL;
	TV :	REAL;
	KI :	REAL;
	KD :	REAL;
END_VAR

VAR
	TX :	REAL;
END_VAR

(*@KEY@: WORKSHEET
NAME: CONTROL_SET2
IEC_LANGUAGE: ST
*)
IF TU > 0.0 AND KS > 0.0 THEN TX := TG / TU / KS; END_IF;
IF pi AND PID THEN
	KP := 0.0;
	TN := 0.0;
	TV := 0.0;
ELSIF PID THEN
	KP := PID_K * TX;
	TN := PID_TN * TU;
	TV := PID_TV * TU;
ELSIF PI THEN
	KP := PI_K * TX;
	TN := PI_TN * TU;
ELSE
	KP := P_K * TX;
END_IF;

(* KI and KD are calculated *)
IF TN > 0.0 THEN KI := KP / TN; ELSE KI := 0.0; END_IF;
KD := KP * TV;

(* revision history
hm	4. nov 2007	rev 1.0
	original version

hm	11. mar. 2009	rev 1.1
	real constants updated to new systax using dot

*)
(*@KEY@: END_WORKSHEET *)
END_FUNCTION_BLOCK

(* ---- COUNT_BR.ST ---- *)
(*@PROPERTIES_EX@
TYPE: POU
LOCALE: 0
IEC_LANGUAGE: ST
PLC_TYPE: independent
PROC_TYPE: independent
GROUP: LOGIC.FF_EDGE_TRIGGERED
*)
(*@KEY@:DESCRIPTION*)
version 1.0	16 jan 2008
programmer 	hugo
tested BY	tobias

Count_R is a byte counter with independen up and dn inputs. the counter counts from 0 to mx and continues at 0 after is has reached mx
a step input sets the counters stepping width.
(*@KEY@:END_DESCRIPTION*)
FUNCTION_BLOCK COUNT_BR

(*Group:Default*)

VAR_INPUT
	SET :	BOOL;
	IN :	BYTE;
	UP :	BOOL;
	DN :	BOOL;
	STEP :	BYTE := BYTE#1;
	MX :	BYTE := BYTE#255;
	RST :	BOOL;
END_VAR

VAR_OUTPUT
	CNT :	BYTE;
END_VAR

VAR
	last_up :	BOOL;
	last_dn :	BOOL;
END_VAR

(*@KEY@: WORKSHEET
NAME: COUNT_BR
IEC_LANGUAGE: ST
*)
IF rst THEN
	cnt := BYTE#0;
ELSIF set THEN
	cnt := INT_TO_BYTE(LIMIT(0,_BYTE_TO_INT(in),_BYTE_TO_INT(mx)));
ELSIF up AND NOT last_up THEN
	cnt := INT_TO_BYTE(inc(_BYTE_TO_INT(cnt),_BYTE_TO_INT(step),_BYTE_TO_INT(mx)));
ELSIF dn AND NOT last_dn THEN
	cnt := INT_TO_BYTE(inc(_BYTE_TO_INT(cnt),_BYTE_TO_INT(step) * -1,_BYTE_TO_INT(mx)));
END_IF;
last_up := up;
last_dn := dn;

(* revision history
hm	16. jan 2008	rev 1.0
	original version

*)
(*@KEY@: END_WORKSHEET *)
END_FUNCTION_BLOCK

(* ---- COUNT_CHAR.ST ---- *)
(*@PROPERTIES_EX@
TYPE: POU
LOCALE: 0
IEC_LANGUAGE: ST
PLC_TYPE: independent
PROC_TYPE: independent
GROUP: STRINGS
*)
(*@KEY@:DESCRIPTION*)
version 1.1	29. mar. 2008
programmer 		kurt
tested by		hugo

COUNT_CHAR how often a character CHAR occurs within a string STR.
(*@KEY@:END_DESCRIPTION*)
FUNCTION_BLOCK COUNT_CHAR

(*Group:Default*)

VAR_INPUT
	STR :	STRING;
	CHR :	BYTE;
END_VAR

VAR_OUTPUT
	COUNT_CHAR :	INT;
END_VAR

VAR
	I :	INT;
	pos :	INT;
END_VAR

(*@KEY@: WORKSHEET
NAME: COUNT_CHAR
IEC_LANGUAGE: ST
*)
I := LEN(str);
COUNT_CHAR := 0;
FOR pos := 1 TO I DO
	IF INT_TO_BYTE(GET_CHAR(str,pos)) = CHR THEN COUNT_CHAR := COUNT_CHAR + 1; END_IF;
END_FOR;

(* revision history
hm	29. feb 2008	rev 1.0
	original version

hm	29. mar. 2008	rev 1.1
	changed STRING to STRING(STRING_LENGTH)
*)
(*@KEY@: END_WORKSHEET *)
END_FUNCTION_BLOCK

(* ---- COUNT_DR.ST ---- *)
(*@PROPERTIES_EX@
TYPE: POU
LOCALE: 0
IEC_LANGUAGE: ST
PLC_TYPE: independent
PROC_TYPE: independent
GROUP: LOGIC.FF_EDGE_TRIGGERED
*)
(*@KEY@:DESCRIPTION*)
version 1.1	20. jan. 2011
programmer 	hugo
tested BY	tobias

Count_DR is a DWORD counter with independen up and dn inputs. the counter counts from 0 to mx and continues at 0 after is has reached mx
a step input sets the counters stepping width.
(*@KEY@:END_DESCRIPTION*)
FUNCTION_BLOCK COUNT_DR

(*Group:Default*)

VAR_INPUT
	SET :	BOOL;
	IN :	DWORD;
	UP :	BOOL;
	DN :	BOOL;
	STEP :	DWORD := DWORD#1;
	MX :	DWORD := DWORD#16#FFFF_FFFF;
	RST :	BOOL;
END_VAR

VAR_OUTPUT
	CNT :	DWORD;
END_VAR

VAR
	CNT2 :	UDINT;
	STEP2 :	UDINT;
	MX2 :	UDINT;
	last_up :	BOOL;
	last_dn :	BOOL;
END_VAR

(*@KEY@: WORKSHEET
NAME: COUNT_DR
IEC_LANGUAGE: ST
*)
STEP2 := DWORD_TO_UDINT(STEP);
MX2   := DWORD_TO_UDINT(MX);
CNT2  := DWORD_TO_UDINT(CNT);

IF rst THEN
	CNT2 := UDINT#0;
ELSIF set THEN
	CNT2 := LIMIT(UDINT#0,DWORD_TO_UDINT(in),mx2);
ELSIF up AND NOT last_up THEN
	IF STEP2 > MX2 - CNT2 THEN
		CNT2 := CNT2 - MX2 + STEP2 - UDINT#1;
	ELSE
		CNT2 := CNT2 + STEP2;
	END_IF;
ELSIF dn AND NOT last_dn THEN
	IF STEP2 > CNT2 THEN
		CNT2 := CNT2 - STEP2 + MX2 + UDINT#1;
	ELSE
		CNT2 := CNT2 - STEP2;
	END_IF;
END_IF;
last_up := up;
last_dn := dn;

CNT := UDINT_TO_DWORD(CNT2);

(* revision history
hm	12. jun 2008	rev 1.0
	original version

hm	20. jan. 2011	rev 1.1
	corrected init value of MX to 16#FFFFFFFF

*)
(*@KEY@: END_WORKSHEET *)
END_FUNCTION_BLOCK

(* ---- COUNT_SUBSTRING.ST ---- *)
(*@PROPERTIES_EX@
TYPE: POU
LOCALE: 0
IEC_LANGUAGE: ST
PLC_TYPE: independent
PROC_TYPE: independent
GROUP: STRINGS
*)
(*@KEY@:DESCRIPTION*)
version 1.0	20. jan. 2011
programmed	kurt
tested by	tobias

count_substring returns the number of occurences of a substring in a string

(*@KEY@:END_DESCRIPTION*)
FUNCTION_BLOCK COUNT_SUBSTRING

(*Group:Default*)

VAR_INPUT
	SEARCH :	STRING;
	STR :	STRING;
END_VAR

VAR_OUTPUT
	COUNT_SUBSTRING :	INT;
END_VAR

VAR
	pos :	INT;
	size :	INT;
END_VAR

(*@KEY@: WORKSHEET
NAME: COUNT_SUBSTRING
IEC_LANGUAGE: ST
*)
COUNT_SUBSTRING := 0;
size := LEN(SEARCH);
REPEAT
   pos := FIND(STR,SEARCH);
   IF pos > 0 THEN
      STR := REPLACE(STR, '', size,pos);
      COUNT_SUBSTRING := COUNT_SUBSTRING + 1;
   END_IF;
UNTIL pos = 0
END_REPEAT;

(* revision history
ks	20. jan. 2011	rev 1.0
	original version

*)

(*@KEY@: END_WORKSHEET *)
END_FUNCTION_BLOCK

(* ---- CPOL.ST ---- *)
(*@PROPERTIES_EX@
TYPE: POU
LOCALE: 0
IEC_LANGUAGE: ST
PLC_TYPE: independent
PROC_TYPE: independent
GROUP: MATHEMATICAL.COMPLEX
*)
(*@KEY@:DESCRIPTION*)
version 1.0	21 feb 2008
programmer 	hugo
tested by	oscat

this function creates a complex numbers for the polar form with the inputs L (length) an A for Angle.
(*@KEY@:END_DESCRIPTION*)
FUNCTION_BLOCK CPOL

(*Group:Default*)

VAR_INPUT
	L :	REAL;
	A :	REAL;
END_VAR

VAR_OUTPUT
	CPOL :	oscat_complex;
END_VAR

(*@KEY@: WORKSHEET
NAME: CPOL
IEC_LANGUAGE: ST
*)
CPOL.re := L * COS(A);
CPOL.im := L * SIN(A);

(* revision history
hm	21. feb 2008	rev 1.0
	original version

*)
(*@KEY@: END_WORKSHEET *)
END_FUNCTION_BLOCK

(* ---- CPOW.ST ---- *)
(*@PROPERTIES_EX@
TYPE: POU
LOCALE: 0
IEC_LANGUAGE: ST
PLC_TYPE: independent
PROC_TYPE: independent
GROUP: MATHEMATICAL.COMPLEX
*)
(*@KEY@:DESCRIPTION*)
version 1.0	21 feb 2008
programmer 	hugo
tested by	oscat

this function calculates the complex power function x to the power of y
(*@KEY@:END_DESCRIPTION*)
FUNCTION_BLOCK CPOW

(*Group:Default*)

VAR_INPUT
	X :	oscat_complex;
	Y :	oscat_complex;
END_VAR

VAR_OUTPUT
	CPOW :	oscat_complex;
END_VAR

VAR
	CLOG :	CLOG;
	CEXP :	CEXP;
	CMUL :	CMUL;
END_VAR

(*@KEY@: WORKSHEET
NAME: CPOW
IEC_LANGUAGE: ST
*)
CLOG(X:=X);
CMUL(X:=Y,Y:=CLOG.CLOG);
CEXP(X:=CMUL.CMUL);
CPOW := CEXP.CEXP;

(* revision history
hm	21. feb 2008	rev 1.0
	original version

*)
(*@KEY@: END_WORKSHEET *)
END_FUNCTION_BLOCK

(* ---- CRC_GEN.ST ---- *)
(*@PROPERTIES_EX@
TYPE: POU
LOCALE: 0
IEC_LANGUAGE: ST
PLC_TYPE: independent
PROC_TYPE: independent
GROUP: LOGIC.OTHER
*)
(*@KEY@:DESCRIPTION*)
version 2.0	16.Jan. 2011
programmer 	hugo
tested by	tobias

CRC_GEN generates a CRC checksum from a block of data and returns  the checksum in a DWORD to be connected to the data for transmission.
the CRC Polynom is specified with the config variable PN and the length of the Polynom is specified by PL
A Polynom x4 + X + 1 is represented by 0011 with length 4, the highest order bit is not specified at all..

(*@KEY@:END_DESCRIPTION*)
FUNCTION_BLOCK CRC_GEN

(*Group:Default*)

VAR_IN_OUT
	PT :	oscat_arb_0_249;
END_VAR

VAR_INPUT
	SIZE :	UINT;
	PL :	UINT;
	PN :	DWORD;
	INIT :	DWORD;
	REV_IN :	BOOL;
	REV_OUT :	BOOL;
	XOR_OUT :	DWORD;
END_VAR

VAR_OUTPUT
	CRC_GEN :	DWORD;
END_VAR

VAR
	pos :	INT;
	shift :	INT;
	dx :	BYTE;
	bits :	INT;
END_VAR

(*@KEY@: WORKSHEET
NAME: CRC_GEN
IEC_LANGUAGE: ST
*)
(* align polygon *)
shift := 32 - UINT_TO_INT(PL);
PN := SHL(PN, shift);

(* load first 4 bytes into register minimum message size is 4 bytes
	for smaller messages fill with 0#s at the beginning*)
FOR pos := 0 TO 3 DO
	IF REV_IN THEN CRC_GEN := SHL(CRC_GEN, 8) OR BYTE_TO_DWORD(REVERSE(PT[pos])); ELSE CRC_GEN := SHL(CRC_GEN, 8) OR BYTE_TO_DWORD(PT[pos]); END_IF;
END_FOR;
pos := 4;

(* xor with init value *)
CRC_GEN := CRC_GEN XOR SHL(init, shift);

(* calculate CRC for each byte *)
WHILE pos < UINT_TO_INT(size) DO
	IF REV_IN THEN DX := REVERSE(PT[pos]); ELSE DX := PT[pos]; END_IF;
	pos := pos + 1;
	(* crc calculation for one byte *)
	FOR bits := 0 TO 7 DO
		IF (CRC_GEN AND DWORD#16#8000_0000) > DWORD#0 THEN (* CRC_GEN.31 *)
			CRC_GEN := (SHL(CRC_GEN, 1) OR BOOL_TO_DWORD((DX AND BYTE#16#80) > BYTE#0)) XOR PN; (* DX.7 *)
		ELSE
			CRC_GEN := SHL(CRC_GEN, 1) OR BOOL_TO_DWORD((DX AND BYTE#16#80) > BYTE#0); (* DX.7 *)
		END_IF;
		dx := SHL(dx, 1);
	END_FOR;
END_WHILE;

(* all bytes are processed, need to finish the registers 32 bits *)
FOR bits := 0 TO 31 DO
	IF (CRC_GEN AND DWORD#16#8000_0000) > DWORD#0 THEN (* CRC_GEN.31 *)
		CRC_GEN := (SHL(CRC_GEN, 1) OR BOOL_TO_DWORD((DX AND BYTE#16#80) > BYTE#0)) XOR PN; (* DX.7 *)
	ELSE
		CRC_GEN := SHL(CRC_GEN, 1) OR BOOL_TO_DWORD((DX AND BYTE#16#80) > BYTE#0); (* DX.7 *)
	END_IF;
END_FOR;

(* final XOR *)
CRC_GEN := SHR(CRC_GEN, shift) XOR XOR_OUT;

(* reverse the crc_out put if necessary *)
IF REV_OUT THEN CRC_GEN := REFLECT(CRC_GEN, UINT_TO_INT(PL)); END_IF;

(* typical crc polynoms

CRC-4-ITU 			x4 + x + 1 					(ITU G.704, p. 12) 	0x3 or 0xC (0x9)
CRC-5-ITU 			x5 + x4 + x2 + 1 			(ITU G.704, p. 9) 	0x15 or 0x15 (0x0B) Bluetooth
CRC-5-USB 			x5 + x2 + 1 				(use: USB token packets) 	0x05 or 0x14 (0x9)
CRC-6-ITU 			x6 + x + 1 					(ITU G.704, p. 3) 	0x03 or 0x30 (0x21)
CRC-7 				x7 + x3 + 1 				(use: telecom systems, MMC) 	0x09 or 0x48 (0x11)
CRC-8-ATM 			x8 + x2 + x + 1 				(use: ATM HEC) 	0x07 or 0xE0 (0xC1)
CRC-8-CCITT 		x8 + x7 + x3 + x2 + 1 		(use: 1-Wire bus) 	0x8D or 0xB1 (0x63)
CRC-8-Dallas/Maxim 	x8 + x5 + x4 + 1 			(use: 1-Wire bus) 	0x31 or 0x8C (0x19)
CRC-8 				x8 + x7 + x6 + x4 + x2 + 1 	0xD5 or 0xAB (0x57)
CRC-8-SAE J1850 	x8 + x4 + x3 + x2 + 1 		0x1D or 0xB8
CRC-10 				x10 + x9 + x5 + x4 + x + 1 	0x233 or 0x331 (0x263)
CRC-12 				x12 + x11 + x3 + x2 + x + 1 (use: telecom systems) 	0x80F or 0xF01 (0xE03)
CRC-15-CAN 			x15 + x14 + x10 + x8 + x7 + x4 + x3 + 1 	0x4599 or 0x4CD1 (0x19A3)
CRC-16-Fletcher 	Not a CRC; see Fletcher's checksum 	Used in Adler-32 A & B CRCs
CRC-16-CCITT 	x16 + x12 + x5 + 1 (XMODEM,X.25, V.41, Bluetooth, PPP, IrDA; known as "CRC-CCITT") 	0x1021 or 0x8408 (0x0811)
CRC-16-IBM 	x16 + x15 + x2 + 1 (USB, many others; also known as "CRC-16") 	0x8005 or 0xA001 (0x4003)
CRC-24-Radix-64 	x24 + x23 + x18 + x17 + x14 + x11 + x10 + x7 + x6 + x5 + x4 + x3 + x + 1 	0x864CFB or 0xDF3261 (0xBE64C3)
CRC-32-Adler 	Not a CRC; see Adler-32 	See Adler-32
CRC-32-MPEG2 	x32 + x26 + x23 + x22 + x16 + x12 + x11 + x10 + x8 + x7 + x5 + x4 + x2 + x + 1 	0x04C11DB7 or 0xEDB88320 (0xDB710641) Also used in IEEE 802.3
CRC-32-IEEE 802.3 	x32 + x26 + x23 + x22 + x16 + x12 + x11 + x10 + x8 + x7 + x5 + x4 + x2 + x + 1 (V.42) 	0x04C11DB7 or 0xEDB88320 (0xDB710641)
CRC-32C (Castagnoli) 	x32 + x28 + x27 + x26 + x25 + x23 + x22 + x20 + x19 + x18 + x14 + x13 + x11 + x10 + x9 + x8 + x6 + 1 	0x1EDC6F41 or 0x82F63B78 (0x05EC76F1)
CRC-64-ISO 	x64 + x4 + x3 + x + 1 (use: ISO 3309) 	0x000000000000001B or 0xD800000000000000 (0xB000000000000001)
CRC-64-ECMA-182 	x64 + x62 + x57 + x55 + x54 + x53 + x52 + x47 + x46 + x45 + x40 + x39 + x38 + x37 + x35 + x33 + x32 + x31 + x29 + x27 + x24 + x23 + x22 + x21 + x19 + x17 + x13 + x12 + x10 + x9 + x7 + x4 + x + 1
(as described in ECMA-182 p.63) 	0x42F0E1EBA9EA3693 or 0xC96C5795D7870F42 (0x92D8AF2BAF0E1E85)
*)

(* revision history

hm	9.6.2007		rev 1.0
	original version

hm	11.9.2007		rev 1.1
	deleted unused variable i

hm	9. oct 2007 	rev 1.2
	added init code for crc and xor_out
	added refelct in and reflect_out (rev_in und Rev_out)

hm	2. jan 2008	rev 1.3
	small changes for performance improvements

hm	16. mar. 2008	rev 1.4
	changed type of input size to uint

hm	10. mar. 2009	rev 1.5
	removed nested comments

hm	16. jan. 2011	rev 2.0
	new version
*)

(*@KEY@: END_WORKSHEET *)
END_FUNCTION_BLOCK

(* ---- CSET.ST ---- *)
(*@PROPERTIES_EX@
TYPE: POU
LOCALE: 0
IEC_LANGUAGE: ST
PLC_TYPE: independent
PROC_TYPE: independent
GROUP: MATHEMATICAL.COMPLEX
*)
(*@KEY@:DESCRIPTION*)
version 1.0	21 feb 2008
programmer 	hugo
tested by	oscat

this function creates a complex number from two real inputs
(*@KEY@:END_DESCRIPTION*)
FUNCTION_BLOCK CSET

(*Group:Default*)

VAR_INPUT
	RE :	REAL;
	IM :	REAL;
END_VAR

VAR_OUTPUT
	CSET :	oscat_complex;
END_VAR

(*@KEY@: WORKSHEET
NAME: CSET
IEC_LANGUAGE: ST
*)
CSET.re := RE;
CSET.im := IM;

(* revision history
hm	21. feb 2008	rev 1.0
	original version

*)
(*@KEY@: END_WORKSHEET *)
END_FUNCTION_BLOCK

(* ---- CSIN.ST ---- *)
(*@PROPERTIES_EX@
TYPE: POU
LOCALE: 0
IEC_LANGUAGE: ST
PLC_TYPE: independent
PROC_TYPE: independent
GROUP: MATHEMATICAL.COMPLEX
*)
(*@KEY@:DESCRIPTION*)
version 1.0	21 feb 2008
programmer 	hugo
tested by	oscat

this function calculates the sinus function of a complex number
(*@KEY@:END_DESCRIPTION*)
FUNCTION_BLOCK CSIN

(*Group:Default*)

VAR_INPUT
	X :	oscat_complex;
END_VAR

VAR_OUTPUT
	CSIN :	oscat_complex;
END_VAR

(*@KEY@: WORKSHEET
NAME: CSIN
IEC_LANGUAGE: ST
*)
CSIN.re := cosH(X.im) * SIN(X.re);
CSIN.im := sinH(X.im) * COS(X.re);

(* revision history
hm	21. feb 2008	rev 1.0
	original version

*)
(*@KEY@: END_WORKSHEET *)
END_FUNCTION_BLOCK

(* ---- CSINH.ST ---- *)
(*@PROPERTIES_EX@
TYPE: POU
LOCALE: 0
IEC_LANGUAGE: ST
PLC_TYPE: independent
PROC_TYPE: independent
GROUP: MATHEMATICAL.COMPLEX
*)
(*@KEY@:DESCRIPTION*)
version 1.0	21 feb 2008
programmer 	hugo
tested by	oscat

this function calculates the sinus function of a complex number
(*@KEY@:END_DESCRIPTION*)
FUNCTION_BLOCK CSINH

(*Group:Default*)

VAR_INPUT
	X :	oscat_complex;
END_VAR

VAR_OUTPUT
	CSINH :	oscat_complex;
END_VAR

(*@KEY@: WORKSHEET
NAME: CSINH
IEC_LANGUAGE: ST
*)
CSINH.re := sinH(X.re) * COS(X.im);
CSINH.im := cosH(X.re) * SIN(X.im);

(* revision history
hm	21. feb 2008	rev 1.0
	original version

*)
(*@KEY@: END_WORKSHEET *)
END_FUNCTION_BLOCK

(* ---- CSQRT.ST ---- *)
(*@PROPERTIES_EX@
TYPE: POU
LOCALE: 0
IEC_LANGUAGE: ST
PLC_TYPE: independent
PROC_TYPE: independent
GROUP: MATHEMATICAL.COMPLEX
*)
(*@KEY@:DESCRIPTION*)
version 1.0	21 feb 2008
programmer 	hugo
tested by	oscat

this function calculates the complex sqare root
(*@KEY@:END_DESCRIPTION*)
FUNCTION_BLOCK CSQRT

(*Group:Default*)

VAR_INPUT
	X :	oscat_complex;
END_VAR

VAR_OUTPUT
	CSQRT :	oscat_complex;
END_VAR

VAR
	temp :	REAL;
END_VAR

(*@KEY@: WORKSHEET
NAME: CSQRT
IEC_LANGUAGE: ST
*)
temp := HYPOT(x.re, x.im);
CSQRT.re :=  SQRT(0.5 * (temp + x.re));
CSQRT.im :=  INT_TO_REAL(sgn(x.im)) * SQRT(0.5 * (temp - x.re));

(* revision history
hm	21. feb 2008	rev 1.0
	original version

*)
(*@KEY@: END_WORKSHEET *)
END_FUNCTION_BLOCK

(* ---- CSUB.ST ---- *)
(*@PROPERTIES_EX@
TYPE: POU
LOCALE: 0
IEC_LANGUAGE: ST
PLC_TYPE: independent
PROC_TYPE: independent
GROUP: MATHEMATICAL.COMPLEX
*)
(*@KEY@:DESCRIPTION*)
version 1.0	21 feb 2008
programmer 	hugo
tested by	oscat

this function subtracts two complex numbers
(*@KEY@:END_DESCRIPTION*)
FUNCTION_BLOCK CSUB

(*Group:Default*)

VAR_INPUT
	X :	oscat_complex;
	Y :	oscat_complex;
END_VAR

VAR_OUTPUT
	CSUB :	oscat_complex;
END_VAR

(*@KEY@: WORKSHEET
NAME: CSUB
IEC_LANGUAGE: ST
*)
CSUB.re := X.re - Y.re;
CSUB.im := X.im - Y.im;

(* revision history
hm	21. feb 2008	rev 1.0
	original version

*)
(*@KEY@: END_WORKSHEET *)
END_FUNCTION_BLOCK

(* ---- CTAN.ST ---- *)
(*@PROPERTIES_EX@
TYPE: POU
LOCALE: 0
IEC_LANGUAGE: ST
PLC_TYPE: independent
PROC_TYPE: independent
GROUP: MATHEMATICAL.COMPLEX
*)
(*@KEY@:DESCRIPTION*)
version 1.1	10. mar. 2009
programmer 	hugo
tested by	oscat

this function calculates the tangens function of a complex number

(*@KEY@:END_DESCRIPTION*)
FUNCTION_BLOCK CTAN

(*Group:Default*)

VAR_INPUT
	X :	oscat_complex;
END_VAR

VAR_OUTPUT
	CTAN :	oscat_complex;
END_VAR

VAR
	temp :	REAL;
	xi2 :	REAL;
	xr2 :	REAL;
END_VAR

(*@KEY@: WORKSHEET
NAME: CTAN
IEC_LANGUAGE: ST
*)
xi2 := 2.0 * x.im;
xr2 := 2.0 * x.re;
temp := 1.0 / (COS(xr2) + COSH( xi2));
CTAN.re := temp * SIN(xr2);
CTAN.im := temp * SINH(xi2);

(* revision history
hm	21. feb 2008	rev 1.0
	original version

hm	10. mar 2009	rev 1.1
	faster code
*)
(*@KEY@: END_WORKSHEET *)
END_FUNCTION_BLOCK

(* ---- CTANH.ST ---- *)
(*@PROPERTIES_EX@
TYPE: POU
LOCALE: 0
IEC_LANGUAGE: ST
PLC_TYPE: independent
PROC_TYPE: independent
GROUP: MATHEMATICAL.COMPLEX
*)
(*@KEY@:DESCRIPTION*)
version 1.1	10. mar. 2009
programmer 	hugo
tested by	oscat

this function calculates the complex hyperbolictangens

(*@KEY@:END_DESCRIPTION*)
FUNCTION_BLOCK CTANH

(*Group:Default*)

VAR_INPUT
	X :	oscat_complex;
END_VAR

VAR_OUTPUT
	CTANH :	oscat_complex;
END_VAR

VAR
	xi2 :	REAL;
	xr2 :	REAL;
	temp :	REAL;
END_VAR

(*@KEY@: WORKSHEET
NAME: CTANH
IEC_LANGUAGE: ST
*)
xi2 := 2.0 * x.im;
xr2 := 2.0 * x.re;
temp := 1.0 /(COSH(xr2) + COS(xi2));
CTANH.re := temp * SINH(xr2);
CTANH.im := temp * SIN(xi2);

(* revision history
hm	21. feb 2008	rev 1.0
	original version

hm	10. mar. 2009	rev 1.1
	new faster code

*)

(*@KEY@: END_WORKSHEET *)
END_FUNCTION_BLOCK

(* ---- CTRL_OUT.ST ---- *)
(*@PROPERTIES_EX@
TYPE: POU
LOCALE: 0
IEC_LANGUAGE: ST
PLC_TYPE: independent
PROC_TYPE: independent
GROUP: ENGINEERING.CONTROL
*)
(*@KEY@:DESCRIPTION*)
version 1.1	3. nov 2008
programmer 	hugo
tested by	oscat
(*@KEY@:END_DESCRIPTION*)
FUNCTION_BLOCK CTRL_OUT

(*Group:Default*)

VAR_INPUT
	CI :	REAL;
	OFFSET :	REAL;
	MAN_IN :	REAL;
	LIM_L :	REAL;
	LIM_H :	REAL;
	MANUAL :	BOOL;
END_VAR

VAR_OUTPUT
	Y :	REAL;
	LIM :	BOOL;
END_VAR

(*@KEY@: WORKSHEET
NAME: CTRL_OUT
IEC_LANGUAGE: ST
*)
Y := SEL(manual, CI, MAN_IN) + OFFSET;

(* Limit the output *)
IF Y >= LIM_H THEN
	Y := LIM_H;
	LIM := TRUE;
ELSIF Y <= lim_L THEN
	Y := LIM_L;
	LIM := TRUE;
ELSE
	LIM := FALSE;
END_IF;

(* revision history
hm 	2. jun. 2008 	rev 1.0
	original version

hm	3. nov. 2008	rev 1.1
	optimized code
*)
(*@KEY@: END_WORKSHEET *)
END_FUNCTION_BLOCK

(* ---- CTRL_PI.ST ---- *)
(*@PROPERTIES_EX@
TYPE: POU
LOCALE: 0
IEC_LANGUAGE: ST
PLC_TYPE: independent
PROC_TYPE: independent
GROUP: ENGINEERING.CONTROL
*)
(*@KEY@:DESCRIPTION*)
version 2.0	30. jun. 2008
programmer 	hugo
tested by	oscat

FT_PI is a PI controller with manual functionality.
The PID controller works according to the fomula Y = e *(KP+ KI * INTEG(e) ) + offset, while e = set_point - actual.
a rst will reset all internal data, while a switch to manual will cause the controller to follow the function Y = manual_in + offset.
limit_h and Limit_l set the possible output range of Y.
the output flags lim will signal that the output limits are active and overflow will signal that the integrator has reached its limits.

since rev 1.1 the "trapezregel is used for more accuracy.
rev 1.2 added selective integratin which means the integrative component is only active within a small range of the target value
this avoids the integrator to go to limits while an input setpoint change happened and is only causing overshoots.
the int_band is by default 100 which means the int is active all the time and if set to for example to 0.1 the integrator is only active
while the input is between 0.9 and 1.1 of the set_point value.

default values for KP = 1, TN = 1, TV = 1, LIMIT_L = -1000, LIMIT_H = +1000.
(*@KEY@:END_DESCRIPTION*)
FUNCTION_BLOCK CTRL_PI

(*Group:Default*)

VAR_INPUT
	ACT :	REAL;
	SET :	REAL;
	SUP :	REAL;
	OFS :	REAL;
	M_I :	REAL;
	MAN :	BOOL;
	RST :	BOOL := FALSE;
	KP :	REAL := 1.0;
	KI :	REAL := 1.0;
	LL :	REAL := -1000.0;
	LH :	REAL := 1000.0;
END_VAR

VAR_OUTPUT
	Y :	REAL;
	DIFF :	REAL;
	LIM :	BOOL;
END_VAR

VAR
	pi :	FT_PIWL;
	co :	CTRL_OUT;
END_VAR

(*@KEY@: WORKSHEET
NAME: CTRL_PI
IEC_LANGUAGE: ST
*)
DIFF := CTRL_IN(SET, ACT, SUP);
pi(in := DIFF, kp := KP, ki := KI, lim_l := LL, lim_h := LH, rst := RST);
co(ci := pi.Y, OFFSET := OFS, man_in := M_I, lim_l := LL, lim_h := LH, manual := MAN);
Y := co.Y;
LIM := co.LIM;

(* revision history
hm 	31.10.2007 	rev 1.0
	original version

hm	3.11.2007	rev 1.1
	added noise input to filter noise
	added output diff
	set limit output false when output is within limits
	overfolw was not set correctly

hm	5. jan 2008	rev 1.2
	improved performance

hm	30. jun. 2008	rev 2.0
	rewritten using new modular approach*)
(*@KEY@: END_WORKSHEET *)
END_FUNCTION_BLOCK

(* ---- CTRL_PID.ST ---- *)
(*@PROPERTIES_EX@
TYPE: POU
LOCALE: 0
IEC_LANGUAGE: ST
PLC_TYPE: independent
PROC_TYPE: independent
GROUP: ENGINEERING.CONTROL
*)
(*@KEY@:DESCRIPTION*)
version 2.0	30. jun. 2008
programmer 	hugo
tested by	oscat

FT_PI is a PI controller with manual functionality.
The PID controller works according to the fomula Y = e *(KP+ KI * INTEG(e) ) + offset, while e = set_point - actual.
a rst will reset all internal data, while a switch to manual will cause the controller to follow the function Y = manual_in + offset.
limit_h and Limit_l set the possible output range of Y.
the output flags lim will signal that the output limits are active.
(*@KEY@:END_DESCRIPTION*)
FUNCTION_BLOCK CTRL_PID

(*Group:Default*)

VAR_INPUT
	ACT :	REAL;
	SET :	REAL;
	SUP :	REAL;
	OFS :	REAL;
	M_I :	REAL;
	MAN :	BOOL;
	RST :	BOOL := FALSE;
	KP :	REAL := 1.0;
	TN :	REAL := 1.0;
	TV :	REAL := 1.0;
	LL :	REAL := -1000.0;
	LH :	REAL := 1000.0;
END_VAR

VAR_OUTPUT
	Y :	REAL;
	DIFF :	REAL;
	LIM :	BOOL;
END_VAR

VAR
	pid :	FT_PIDWL;
	co :	CTRL_OUT;
END_VAR

(*@KEY@: WORKSHEET
NAME: CTRL_PID
IEC_LANGUAGE: ST
*)
DIFF := CTRL_IN(SET, ACT, SUP);
pid(in := DIFF, kp := KP, tn := TN, tv := TV, lim_l := LL, lim_h := LH, rst := RST);
co(ci := pid.Y, OFFSET := OFS, man_in := M_I, lim_l := LL, lim_h := LH, manual := MAN);
Y := co.Y;
LIM := co.LIM;

(* revision history
hm 	31.10.2007 		rev 1.0
	original version

hm	3.11.2007		rev 1.1
	added noise input to filter noise
	added output diff
	set limit output false when output is within limits
	overfolw was not set correctly

hm	5. jan 2008		rev 1.2
	improved performance

hm	30. jun. 2008	rev 2.0
	rewritten using new modular approach

*)
(*@KEY@: END_WORKSHEET *)
END_FUNCTION_BLOCK

(* ---- CTRL_PWM.ST ---- *)
(*@PROPERTIES_EX@
TYPE: POU
LOCALE: 0
IEC_LANGUAGE: ST
PLC_TYPE: independent
PROC_TYPE: independent
GROUP: ENGINEERING.CONTROL
*)
(*@KEY@:DESCRIPTION*)
version 1.1	21. oct. 2008
programmer 	hugo
tested by	oscat
(*@KEY@:END_DESCRIPTION*)
FUNCTION_BLOCK CTRL_PWM

(*Group:Default*)

VAR_INPUT
	CI :	REAL;
	MAN_IN :	REAL;
	MANUAL :	BOOL;
	F :	REAL;
END_VAR

VAR_OUTPUT
	Q :	BOOL;
END_VAR

VAR
	PW :	PWM_DC;
END_VAR

(*@KEY@: WORKSHEET
NAME: CTRL_PWM
IEC_LANGUAGE: ST
*)
PW(F := F, DC := SEL(MANUAL,CI,MAN_IN));
Q := PW.Q;

(* revision history
hm 	3. jun. 2008 	rev 1.0
	original version

hm	21. oct. 2008	rev 1.1
	optimized code
*)
(*@KEY@: END_WORKSHEET *)
END_FUNCTION_BLOCK

(* ---- CYCLE_4.ST ---- *)
(*@PROPERTIES_EX@
TYPE: POU
LOCALE: 0
IEC_LANGUAGE: ST
PLC_TYPE: independent
PROC_TYPE: independent
GROUP: LOGIC.GENERATORS
*)
(*@KEY@:DESCRIPTION*)
version 1.0
programmer 	hugo
tested by	oscat
(*@KEY@:END_DESCRIPTION*)
FUNCTION_BLOCK CYCLE_4

(*Group:Default*)

VAR_INPUT
	E :	BOOL := TRUE;
	T0 :	TIME;
	T1 :	TIME;
	T2 :	TIME;
	T3 :	TIME;
	S0 :	BOOL;
	SX :	INT;
	SL :	BOOL;
END_VAR

VAR_OUTPUT
	STATE :	INT;
END_VAR

VAR
	tx :	TIME;
	last :	TIME;
	init :	BOOL;
	T_PLC_MS :	T_PLC_MS;
END_VAR

(*@KEY@: WORKSHEET
NAME: CYCLE_4
IEC_LANGUAGE: ST
*)
(* read system *)
T_PLC_MS();
tx:= UDINT_TO_TIME(T_PLC_MS.T_PLC_MS);

(* init on first cycle *)
IF NOT init THEN
	init := TRUE;
	last := tx;
END_IF;

IF E THEN
	IF SL THEN
		(* when sx > 0 then the state sx is forced to start *)
		state:= LIMIT(0,SX,3);
		last := tx;
		(* this is to avoid to reset sx from the calling programm it does work fine on codesys but i am not sure about other systems, because we are writing to an input *)
		SL := FALSE;
	ELSE
		CASE state OF
			0 :	(* wait for T0 and switch to next cycle *)
				IF tx - last >= T0 THEN
					state := 1;
					last := tx;
				END_IF;
			1 : (* wait for T1 over 1st cycle *)
				IF tx - last >= T1 THEN
					state := 2;
					last := tx;
				END_IF;
			2 : (* wait for T1 over 1st cycle *)
				IF tx - last >= T2 THEN
					state := 3;
					last := tx;
				END_IF;
			3 : (* wait for T2 over 2nd cycle *)
				IF tx - last >= T3 THEN
					IF S0 THEN State := 0; END_IF; (* if S0 is false, the sequence stops at state 3 *)
					last := tx;
				END_IF;
		END_CASE;
	END_IF;
ELSE
	state := 0;
	last := tx;
END_IF;

(*
hm	3. nov. 2008	rev 1.0
	original version

*)
(*@KEY@: END_WORKSHEET *)
END_FUNCTION_BLOCK

(* ---- CYCLE_TIME.ST ---- *)
(*@PROPERTIES_EX@
TYPE: POU
LOCALE: 0
IEC_LANGUAGE: ST
PLC_TYPE: independent
PROC_TYPE: independent
GROUP: ENGINEERING.MEASUREMENTS
*)
(*@KEY@:DESCRIPTION*)
version 1.2	16 sep 2007
programmer 	hugo
tested BY	hans

this function block measures the cycle time and displays the last, min and max cycle time of the current task.
the resolution is 1ms.
the cycles output is a dword counter which counts the cycles.
a rst pulse on the input will reset all data.
(*@KEY@:END_DESCRIPTION*)
FUNCTION_BLOCK CYCLE_TIME

(*Group:Default*)

VAR_INPUT
	RST :	BOOL;
END_VAR

VAR_OUTPUT
	CT_MIN :	TIME := t#0s;
	CT_MAX :	TIME := t#0s;
	CT_LAST :	TIME;
	SYSTIME :	TIME;
	SYSDAYS :	INT;
	CYCLES :	DWORD;
END_VAR

VAR
	last_cycle :	TIME;
	tx :	TIME;
	init :	BOOL;
	T_PLC_MS :	T_PLC_MS;
END_VAR

(*@KEY@: WORKSHEET
NAME: CYCLE_TIME
IEC_LANGUAGE: ST
*)
T_PLC_MS();
tx:= UDINT_TO_TIME(T_PLC_MS.T_PLC_MS) - last_cycle;

IF rst THEN
	ct_min := t#10h;
	ct_max := t#0ms;
	cycles := DWORD#0;
ELSIF last_cycle > t#0s THEN
	IF tx < ct_min THEN ct_min := tx;
	ELSIF tx > ct_max THEN ct_max := tx;
	END_IF;
	ct_last := tx;
ELSIF ct_min = t#0s THEN
	ct_min := t#0s - t#1ms;
END_IF;
IF init THEN
	systime := systime + tx;
		IF systime >= t#1d THEN
			systime := systime - t#1d;
			sysdays := sysdays + 1;
		END_IF;
END_IF;
init := TRUE;
last_cycle := last_cycle + tx;
cycles := UDINT_TO_DWORD(DWORD_TO_UDINT(cycles) + UDINT#1);

(*	revision history
hm 12.12.2006		rev 1.1
	added cycles output, a dword cycle counter.
hm 10.3.2007			rev 1.2
	changed initialization of ct_min to t#10h for compatibility with siemens s7

hm	16.9.2007		rev 1.2
	changed Time() in T_PLC_MS() for compatibility resons

*)
(*@KEY@: END_WORKSHEET *)
END_FUNCTION_BLOCK

(* ---- D_TRIG.ST ---- *)
(*@PROPERTIES_EX@
TYPE: POU
LOCALE: 0
IEC_LANGUAGE: ST
PLC_TYPE: independent
PROC_TYPE: independent
GROUP: LOGIC.GENERATORS
*)
(*@KEY@:DESCRIPTION*)
version 1.1	19. feb 2008
programmer 	hugo
tested by	tobias

this block is similar to the IEC Standard R_trig and F_trig but it monitors a DWORD, WORD or Byte Variable instead and generated an Output Pulse for one cycle only when the input has changed.
an additional output x (Dword) will state the chage of the input.
Example: the input has chaged from 0001 to 0010 then the output x will be 2.
(*@KEY@:END_DESCRIPTION*)
FUNCTION_BLOCK D_TRIG

(*Group:Default*)

VAR_INPUT
	IN :	DWORD;
END_VAR

VAR_OUTPUT
	Q :	BOOL;
	X :	DWORD;
END_VAR

VAR
	last_in :	DWORD;
END_VAR

(*@KEY@: WORKSHEET
NAME: D_TRIG
IEC_LANGUAGE: ST
*)
Q := in <> last_in;
X := UDINT_TO_DWORD(DWORD_TO_UDINT(in) - DWORD_TO_UDINT(last_in));
last_in := in;

(* revision history

hm 	4.09.2007		rev 1.0
	original version released

hm	19. feb. 2008	rev 1.1
	performance improvement
*)
(*@KEY@: END_WORKSHEET *)
END_FUNCTION_BLOCK

(* ---- DATE_TO_STRING.ST ---- *)
(*@PROPERTIES_EX@
TYPE: POU
LOCALE: 0
IEC_LANGUAGE: ST
PLC_TYPE: independent
PROC_TYPE: independent
GROUP: EMULATION
*)
(*@KEY@:DESCRIPTION*)

(*@KEY@:END_DESCRIPTION*)
FUNCTION_BLOCK DATE_TO_STRING

(*Group:Default*)

VAR_INPUT
	IDATE :	UDINT;
END_VAR

VAR_OUTPUT
	DATE_STRING :	STRING;
END_VAR

VAR
	st_tmp1 :	STRING;
END_VAR

(*@KEY@: WORKSHEET
NAME: DATE_TO_STRING
IEC_LANGUAGE: ST
*)
st_tmp1 := CONCAT(INT_TO_STRING(YEAR_OF_DATE(IDATE),'%04d-'),INT_TO_STRING(MONTH_OF_DATE(IDATE),'%02d-'));
DATE_STRING := CONCAT(st_tmp1,INT_TO_STRING(day_of_month(IDATE),'%02d'));
(*@KEY@: END_WORKSHEET *)
END_FUNCTION_BLOCK

(* ---- DCF77.ST ---- *)
(*@PROPERTIES_EX@
TYPE: POU
LOCALE: 0
IEC_LANGUAGE: ST
PLC_TYPE: independent
PROC_TYPE: independent
GROUP: TIME_DATE
*)
(*@KEY@:DESCRIPTION*)
version 1.10	7. oct. 2008
programmer 	hugo
tested by	oscat

this is a decoder for a DCF77 signal.
the decoder decodes the DCF77 signal and checks for a valid Date_Time.
since the dcf77 signal is only secured with a simple parity the decoder waits for two consecutive valid transmissions before it sets the output signals.
given a valid reception by the receiver the decoder can take up to 3 minutes to start its clocks the first time.
after a valid signal is detected the error output goes low and dignals a valid dcf signal from the receiver.
a tp is only valid for one program cycle to allow for external rtc setting.
after a valid signal is detected two independent internal clocks are started (RTC and RTC1), the seconds  of these clocks are generated by software since the dcf signal is only valid for minutes.
rtc is always utc ( world time) and rtc1 can be set to any time zone by setting the time_zone_offset and enabling dst for automatic summertime.
a sync output signals the the rtc and rtc1 are in sync with the dcf77 signal, if the dcf77 signal is lost for more then the sync time the sync output goes low
but the rtc and rtc1 outputs keep running based on software timing until a valid dcf77 signal is received again and triggers the clock.
in addition a millisecond output gives further resolutionof the clocks.
a dst output shows if daylight saving time is enables and the weekday output shows which day of week currently is ( 1= monday ... 7= sunday).
(*@KEY@:END_DESCRIPTION*)
FUNCTION_BLOCK DCF77

(*Group:Default*)

VAR_INPUT
	REC :	BOOL;
	SET :	BOOL;
	SDT :	UDINT;
	DSI :	BOOL;
	SYNC_TIMEOUT :	TIME := t#2m;
	TIME_OFFSET :	INT := 1;
	DST_EN :	BOOL := TRUE;
END_VAR

VAR_OUTPUT
	TP :	BOOL;
	DS :	BOOL;
	WDAY :	INT;
	ERROR :	BOOL := TRUE;
	RTC :	UDINT;
	RTC1 :	UDINT;
	MSEC :	INT;
	SYNC :	BOOL;
END_VAR

VAR
	MEZ :	UDINT;
	UTC :	UDINT;
	state :	INT;
	edge :	BOOL;
	tx :	TIME;
	ty :	TIME;
	last :	TIME;
	bits :	oscat_dcf77_bits;
	cnt :	INT;
	i :	INT;
	old_time :	UDINT;
	minute :	INT;
	hour :	INT;
	day :	INT;
	month :	INT;
	year :	INT;
	last_sync :	TIME;
	t1 :	TIME;
	tz :	TIME;
	init :	BOOL;
	word_temp :	WORD;
	bool_temp :	BOOL;
	T_PLC_MS :	T_PLC_MS;
END_VAR

(*@KEY@: WORKSHEET
NAME: DCF77
IEC_LANGUAGE: ST
*)
(* if tp was set it should only be active for 1 cycle *)
TP := FALSE;

(* read system time *)
T_PLC_MS();
t1:= UDINT_TO_TIME(T_PLC_MS.T_PLC_MS);
tx := t1 - last;

IF rec XOR edge THEN
	edge := rec;
	IF NOT rec AND tx > t#1700ms AND tx < t#2000ms THEN
		(* start condition reached *)
		state := 0;
		tp := NOT error;
	ELSIF NOT rec AND tx > t#700ms AND tx < t#1000ms THEN
		(* second switch detected *)
		IF state < 58 THEN state := state +1; ELSE state := 0; END_IF;
	ELSIF rec AND tx  < t#120ms THEN
		(* bit 0 detected  *)
		bits[state] := FALSE;
	ELSIF rec AND tx > t#120ms AND tx < t#250ms THEN
		(* bit 1 detected *)
		bits[state] := TRUE;
	ELSE
		(* error condition received signal is not valid *)
		error := TRUE;
		state := 0;
	END_IF;
	last := last + tx;
	IF rec AND state = 58 THEN
		error := FALSE;

		(* decode the bits and check for possible errors *)
		IF bits[0] OR NOT (bits[17] XOR bits[18]) OR NOT bits[20] THEN error := TRUE; END_IF;
		(* decode minute *)
        word_temp := WORD#0;

        bool_temp:=bits[21];
        word_temp:=BIT_LOAD_W(word_temp,bool_temp,0);    (* word_temp.X0 := bits[21]; *)
        bool_temp:=bits[22];
        word_temp:=BIT_LOAD_W(word_temp,bool_temp,1);    (* word_temp.X1 := bits[22]; *)
        bool_temp:=bits[23];
        word_temp:=BIT_LOAD_W(word_temp,bool_temp,2);    (* word_temp.X2 := bits[23]; *)
        bool_temp:=bits[24];
        word_temp:=BIT_LOAD_W(word_temp,bool_temp,3);    (* word_temp.X3 := bits[24]; *)

        minute := WORD_TO_INT(word_temp);
		IF bits[25] THEN minute := minute +10; END_IF;
		IF bits[26] THEN minute := minute +20; END_IF;
		IF bits[27] THEN minute := minute +40; END_IF;
		IF minute > 59 OR (bits[21] XOR bits[22] XOR bits[23] XOR bits[24] XOR bits[25] XOR bits[26] XOR bits[27] XOR bits[28]) THEN error := TRUE; END_IF;

		(* decode hour *)
        word_temp := WORD#0;

        bool_temp:=bits[29];
        word_temp:=BIT_LOAD_W(word_temp,bool_temp,0);    (* word_temp.X0 := bits[29]; *)
        bool_temp:=bits[30];
        word_temp:=BIT_LOAD_W(word_temp,bool_temp,1);    (* word_temp.X1 := bits[30]; *)
        bool_temp:=bits[31];
        word_temp:=BIT_LOAD_W(word_temp,bool_temp,2);    (* word_temp.X2 := bits[31]; *)
        bool_temp:=bits[32];
        word_temp:=BIT_LOAD_W(word_temp,bool_temp,3);    (* word_temp.X3 := bits[32]; *)

        hour := WORD_TO_INT(word_temp);
		IF bits[33] THEN hour := hour +10; END_IF;
		IF bits[34] THEN hour := hour +20; END_IF;
		IF hour > 23 OR (bits[29] XOR bits[30] XOR bits[31] XOR bits[32] XOR bits[33] XOR bits[34] XOR bits[35]) THEN error := TRUE; END_IF;

		(* decode day of month *)
        word_temp := WORD#0;

        bool_temp:=bits[36];
        word_temp:=BIT_LOAD_W(word_temp,bool_temp,0);    (* word_temp.X0 := bits[36]; *)
        bool_temp:=bits[37];
        word_temp:=BIT_LOAD_W(word_temp,bool_temp,1);    (* word_temp.X1 := bits[37]; *)
        bool_temp:=bits[38];
        word_temp:=BIT_LOAD_W(word_temp,bool_temp,2);    (* word_temp.X2 := bits[38]; *)
        bool_temp:=bits[39];
        word_temp:=BIT_LOAD_W(word_temp,bool_temp,3);    (* word_temp.X3 := bits[39]; *)

        day := WORD_TO_INT(word_temp);
		IF bits[40] THEN day := day + 10; END_IF;
		IF bits[41] THEN day := day + 20; END_IF;
		IF day > 31 THEN error := TRUE; END_IF;

		(* decode day of week *)
        word_temp := WORD#0;

        bool_temp:=bits[42];
        word_temp:=BIT_LOAD_W(word_temp,bool_temp,0);    (* word_temp.X0 := bits[42]; *)
        bool_temp:=bits[43];
        word_temp:=BIT_LOAD_W(word_temp,bool_temp,1);    (* word_temp.X1 := bits[43]; *)
        bool_temp:=bits[44];
        word_temp:=BIT_LOAD_W(word_temp,bool_temp,2);    (* word_temp.X2 := bits[44]; *)

        wday := WORD_TO_INT(word_temp);
		IF wday > 7 OR wday < 1 THEN error := TRUE; END_IF;

		(* decode month *)
        word_temp := WORD#0;

        bool_temp:=bits[45];
        word_temp:=BIT_LOAD_W(word_temp,bool_temp,0);    (* word_temp.X0 := bits[45]; *)
        bool_temp:=bits[46];
        word_temp:=BIT_LOAD_W(word_temp,bool_temp,1);    (* word_temp.X1 := bits[46]; *)
        bool_temp:=bits[47];
        word_temp:=BIT_LOAD_W(word_temp,bool_temp,2);    (* word_temp.X2 := bits[47]; *)
        bool_temp:=bits[48];
        word_temp:=BIT_LOAD_W(word_temp,bool_temp,3);    (* word_temp.X3 := bits[48]; *)

        month := WORD_TO_INT(word_temp);
		IF bits[49] THEN month := month +10; END_IF;
		IF month > 12 THEN error := TRUE; END_IF;

		(* decode year *)
        word_temp := WORD#0;

        bool_temp:=bits[50];
        word_temp:=BIT_LOAD_W(word_temp,bool_temp,0);    (* word_temp.X0 := bits[50]; *)
        bool_temp:=bits[51];
        word_temp:=BIT_LOAD_W(word_temp,bool_temp,1);    (* word_temp.X1 := bits[51]; *)
        bool_temp:=bits[52];
        word_temp:=BIT_LOAD_W(word_temp,bool_temp,2);    (* word_temp.X2 := bits[52]; *)
        bool_temp:=bits[53];
        word_temp:=BIT_LOAD_W(word_temp,bool_temp,3);    (* word_temp.X3 := bits[53]; *)

        year := WORD_TO_INT(word_temp);
		IF bits[54] THEN year := year + 10; END_IF;
		IF bits[55] THEN year := year + 20; END_IF;
		IF bits[56] THEN year := year + 40; END_IF;
		IF bits[57] THEN year := year + 80; END_IF;

		(* check parity for bits 36 to 58 *)
		cnt := 0;
		FOR i := 36 TO 58 DO IF bits[i] THEN cnt := cnt + 1; END_IF; END_FOR;
		IF NOT even(INT_TO_DINT(cnt)) THEN error := TRUE; END_IF;

		(* time must be valid for two cycles to clear error flag *)
		IF NOT error THEN
			(* set outputs *)
			old_time := mez;
			IF year >= 70 THEN year := year + 1900; ELSE year := year + 2000; END_IF;
			mez := set_DT(year,month,day,hour,minute,0);
			DS := bits[17];
			IF DS THEN
				UTC := mez - UDINT#7200;
			ELSE
				UTC := mez - UDINT#3600;
			END_IF;

			(* set trigger signal only if the receiver has received 2 successive minutes *)
			IF mez <> old_time + TIME_TO_UDINT(t#1m) THEN error := TRUE ; END_IF;
		END_IF;
	END_IF;
END_IF;

(* this portion implements a free running clock which is triggered by the dcf77 signal *)
tz := UDINT_TO_TIME(_INT_TO_UDINT(ABS(time_offset))* UDINT#3600000);

(* input sdt is copied to utc at first power up *)
IF NOT init OR SET THEN
	init := TRUE;
	utc := sdt;
	tp := TRUE;
	DS := DSI;
END_IF;

IF tp THEN
	rtc := utc;
	IF DS AND dst_en THEN
		IF time_offset < 0 THEN
        	rtc1 := rtc - TIME_TO_UDINT(tz + t#1h);
        ELSE
            rtc1 := rtc + TIME_TO_UDINT(tz + t#1h);
        END_IF;
	ELSE
		IF time_offset < 0 THEN
            rtc1 := rtc - TIME_TO_UDINT(tz);
        ELSE
            rtc1 := rtc + TIME_TO_UDINT(tz);
        END_IF;
	END_IF;
	sync := TRUE;
	last_sync := last;
	ty := last;
ELSIF rtc > UDINT#0 AND T1 - ty >= t#1s THEN
	rtc := rtc + TIME_TO_UDINT(t#1s);
	rtc1 := rtc1 + TIME_TO_UDINT(t#1s);
	ty := ty + t#1s;
	sync := ty - last_sync < sync_timeout AND last_sync > t#0s;
	wday := DAY_OF_WEEK(DT_TO_DATE(rtc1));
	DS := dst_en AND DST(utc);
END_IF;
msec := TIME_TO_INT(t1 - ty);

(* decode information
bits		content
0			Bitwert immer 0
1 bis 14	reserviert für Betriebsinformationen (nicht für DCF77-Nutzer bestimmt)
15			Rufbit für Alarmierung der PTB-Mitarbeiter
			(bis Mai 2003: Bitwert = 0 falls normale Antenne in Verwendung; 1 = Backupantenne)
16			Bitwert = 1 falls ein Wechsel von MEZ nach MESZ oder umgekehrt bevorsteht; Dauer der Anzeige: 1 Stunde
17 + 18	gültige Zeit = MEZ, falls Bit 17=0 und Bit 18=1
			gültige Zeit = MESZ, falls Bit 17=1 und Bit 18=0
19			Bitwert = 1 falls innerhalb den nächsten 59 Minuten eine Schaltsekunde angeordnet ist. Beim Einfügen einer Schaltsekunde wird anstelle der 59. die 60. Sekundenmarke weggelassen und in der 58. erfolgt ausnahmsweise ein Trägerabfall.
20			Startbit für Zeitinformation (immer 1)
21 - 27		1, 2, 4, 8, 10, 20, 40 Minuten (bitweise Addition)
28			Prüfbit (gerade Parität) für die Bits 21-27
29 - 34		1, 2, 4, 8, 10, 20 Stunden (bitweise Addition)
35			Prüfbit (gerade Parität) für die Bits 29-34
36 - 41		Tagesnummer im aktuellen Monat: 1, 2, 4, 8, 10, 20 (bitweise Addition)
42 - 44		Tagesnummer in der aktuellen Woche: 1, 2, 4 (bitweise Addition)
45 - 49		Monatsnummer: 1, 2, 4, 8, 10 (bitweise Addition)
50 - 57		Jahr (zweistellig): 1, 2, 4, 8, 10, 20, 40, 80 (bitweise Addition)
58			Prüfbit (gerade Parität) füR die Bits 36-57

*)
(* revision history

hm 2.feb 2007		rev 1.1
	change wday and dst outputs when there is no dcf reception

hm	26.feb 2007		rev 1.2
	changed statements where t#1h would be substracted from DT.
	under certain conditions the compiler would crash translating this statement

hm	17. sep 2007	rev 1.3
	replaced time() with T_PLC_MS() for compatibility reasons

hm	24. oct 2007		rev 1.4
	changed dst calculation because function dst was upgraded no error in DCF77 only a change in DST

hm	12. nov 2007		rev 1.5
	changed time_offset from time to integer to allow for negative offset time zones

hm	8. dec 2007		rev 1.6
	corrected an error in time_zone calculation

hm 23. jan 2008		rev 1.7
	added sdt input which is used to initialize rtc and rtc1 during first cycle.

hm 16. mar 2008		rev 1.8
	changed output weekday to wday and dst to ds for compatibility reasons

hm	19. apr. 2008	rev 1.9
	added input dsi to allow to set daylight savings time when SDT is TRUE.
	added asynchronous SET input

hm	7. oct. 2008	rev 1.10
	changed function weekday to day_of_week

*)
(*@KEY@: END_WORKSHEET *)
END_FUNCTION_BLOCK

(* ---- DEAD_BAND_A.ST ---- *)
(*@PROPERTIES_EX@
TYPE: POU
LOCALE: 0
IEC_LANGUAGE: ST
PLC_TYPE: independent
PROC_TYPE: independent
GROUP: ENGINEERING.CONTROL
*)
(*@KEY@:DESCRIPTION*)
version 1.1	11. mar. 2009
programmer 	hugo
tested by	oscat

DEAD_BAND ist eine lineare Übertragungsfunktion mit Totzone. Die Funktion verschiebt den positiven Teil der Kurve um -L und den negativen Teil der Kurve um +L.
DEAD_BAND = X wenn Abs(X) > L wenn Abs(X) > L
DEAD_BAND = 0 wenn Abs(X) <= L
Die Breite der Totzone wird automatisch aus dem Signalrauschen errechnet.

(*@KEY@:END_DESCRIPTION*)
FUNCTION_BLOCK DEAD_BAND_A

(*Group:Default*)

VAR_INPUT
	X :	REAL;
	T :	TIME;
	KL :	REAL := 1.0;
	LM :	REAL;
END_VAR

VAR_OUTPUT
	Y :	REAL;
	L :	REAL;
END_VAR

VAR
	tp1 :	FT_PT1;
	tp2 :	FT_PT1;
END_VAR

(*@KEY@: WORKSHEET
NAME: DEAD_BAND_A
IEC_LANGUAGE: ST
*)
(* filter the input signal *)
tp1(in := X, T:= T);

(* filter the HF portion to generate a stable L *)
tp2(in := ABS(tp1.out - X), T := MULTIME(T, 4.0));

(* now we determine L which is half the width of the dead band *)
L := MIN(KL * tp2.out, LM);

IF X > L THEN
	Y := X - L;
ELSIF X < -L THEN
	Y := X + L;
ELSE
	Y := 0.0;
END_IF;

(* revision history
hm	14. jun. 2008	rev 1.0
	original version

hm	11. mar. 2009	rev 1.1
	real constants updated to new systax using dot

*)
(*@KEY@: END_WORKSHEET *)
END_FUNCTION_BLOCK

(* ---- DEAD_ZONE2.ST ---- *)
(*@PROPERTIES_EX@
TYPE: POU
LOCALE: 0
IEC_LANGUAGE: ST
PLC_TYPE: independent
PROC_TYPE: independent
GROUP: ENGINEERING.CONTROL
*)
(*@KEY@:DESCRIPTION*)
version 1.1	11. mar. 2009
programmer 	hugo
tested by	tobias

dead_zone2 is a linear transfer function which follows a linear function except for x is close to 0.
Y = X if abs(x) > L.
for values of 0 +/- L a hysteresis function will hold the output at + or - L.

(*@KEY@:END_DESCRIPTION*)
FUNCTION_BLOCK DEAD_ZONE2

(*Group:Default*)

VAR_INPUT
	X :	REAL;
	L :	REAL;
END_VAR

VAR_OUTPUT
	Y :	REAL;
END_VAR

(*@KEY@: WORKSHEET
NAME: DEAD_ZONE2
IEC_LANGUAGE: ST
*)
IF ABS(x) > L THEN
	Y := X;
ELSIF Y > 0.0 THEN
	Y := L;
ELSE
	Y := -L;
END_IF;

(* revision history

hm	12. feb. 2007	rev 1.0
	original version

hm	11. mar. 2009	rev 1.1
	real constants updated to new systax using dot

*)

(*@KEY@: END_WORKSHEET *)
END_FUNCTION_BLOCK

(* ---- DEC_2.ST ---- *)
(*@PROPERTIES_EX@
TYPE: POU
LOCALE: 0
IEC_LANGUAGE: ST
PLC_TYPE: independent
PROC_TYPE: independent
GROUP: LOGIC.GATE_LOGIC
*)
(*@KEY@:DESCRIPTION*)
version 1.1	3 Mar 2007
programmer 	hugo
tested by	tobias

a bit input will be decoded to the two outputs Q0 or Q1
dependent on the value of A
A=0 decodes to Q0 and A=1 decodes to Q1
(*@KEY@:END_DESCRIPTION*)
FUNCTION_BLOCK DEC_2

(*Group:Default*)

VAR_INPUT
	D :	BOOL;
	A :	BOOL;
END_VAR

VAR_OUTPUT
	Q0 :	BOOL;
	Q1 :	BOOL;
END_VAR

(*@KEY@: WORKSHEET
NAME: DEC_2
IEC_LANGUAGE: ST
*)
Q0 := D AND NOT A;
Q1 := D AND A;

(* revision history
hm 3.3.2007	rev 1.1
	rewritten in ST for better compatibility
*)
(*@KEY@: END_WORKSHEET *)
END_FUNCTION_BLOCK

(* ---- DEC_4.ST ---- *)
(*@PROPERTIES_EX@
TYPE: POU
LOCALE: 0
IEC_LANGUAGE: ST
PLC_TYPE: independent
PROC_TYPE: independent
GROUP: LOGIC.GATE_LOGIC
*)
(*@KEY@:DESCRIPTION*)
version 1.1	3 Mar 2007
programmer 	hugo
tested by	tobias

a bit input will be decoded to one of the 4 outputs
dependent on the Adress on A0 and A1
(*@KEY@:END_DESCRIPTION*)
FUNCTION_BLOCK DEC_4

(*Group:Default*)

VAR_INPUT
	D :	BOOL;
	A0 :	BOOL;
	A1 :	BOOL;
END_VAR

VAR_OUTPUT
	Q0 :	BOOL;
	Q1 :	BOOL;
	Q2 :	BOOL;
	Q3 :	BOOL;
END_VAR

(*@KEY@: WORKSHEET
NAME: DEC_4
IEC_LANGUAGE: ST
*)
Q0 := D AND NOT A0 AND NOT A1;
Q1 := D AND A0 AND NOT A1;
Q2 := D AND NOT A0 AND A1;
Q3 := D AND A0 AND A1;

(* revision history
hm 3.3.2007	rev 1.1
	rewritten in ST for better compatibility

*)
(*@KEY@: END_WORKSHEET *)
END_FUNCTION_BLOCK

(* ---- DEC_8.ST ---- *)
(*@PROPERTIES_EX@
TYPE: POU
LOCALE: 0
IEC_LANGUAGE: ST
PLC_TYPE: independent
PROC_TYPE: independent
GROUP: LOGIC.GATE_LOGIC
*)
(*@KEY@:DESCRIPTION*)
version 1.3	28. mar. 2009
programmer 	hugo
tested by	oscat

a bit input will be decoded to one of the 8 outputs
dependent on the Adress on A0, A1 and A2

(*@KEY@:END_DESCRIPTION*)
FUNCTION_BLOCK DEC_8

(*Group:Default*)

VAR_INPUT
	D :	BOOL;
	A0 :	BOOL;
	A1 :	BOOL;
	A2 :	BOOL;
END_VAR

VAR_OUTPUT
	Q0 :	BOOL;
	Q1 :	BOOL;
	Q2 :	BOOL;
	Q3 :	BOOL;
	Q4 :	BOOL;
	Q5 :	BOOL;
	Q6 :	BOOL;
	Q7 :	BOOL;
END_VAR

VAR
	X :	BYTE;
END_VAR

(*@KEY@: WORKSHEET
NAME: DEC_8
IEC_LANGUAGE: ST
*)
X:=BIT_LOAD_B(X,A0,0); (* X.0 := A0; *)
X:=BIT_LOAD_B(X,A1,1); (* X.1 := A1; *)
X:=BIT_LOAD_B(X,A2,2); (* X.2 := A2; *)

Q0 := FALSE;
Q1 := FALSE;
Q2 := FALSE;
Q3 := FALSE;
Q4 := FALSE;
Q5 := FALSE;
Q6 := FALSE;
Q7 := FALSE;

CASE _BYTE_TO_INT(X) OF
	0 : Q0 := D;
	1 : Q1 := D;
	2 : Q2 := D;
	3 : Q3 := D;
	4 : Q4 := D;
	5 : Q5 := D;
	6 : Q6 := D;
	7 : Q7 := D;
END_CASE;

(* revision history
hm 3. mar. 2007	rev 1.1
	rewritten in ST for better compatibility

hm	26. oct. 2008	rev 1.2
	code optimized

hm	28. mar. 2009	rev 1.3
	replaced multiple assignments
*)
(*@KEY@: END_WORKSHEET *)
END_FUNCTION_BLOCK

(* ---- DEC_TO_BYTE.ST ---- *)
(*@PROPERTIES_EX@
TYPE: POU
LOCALE: 0
IEC_LANGUAGE: ST
PLC_TYPE: independent
PROC_TYPE: independent
GROUP: STRINGS
*)
(*@KEY@:DESCRIPTION*)
version 1.1	30. sep 2008
programmer 	hugo
tested by	oscat

DEC_TO_byte converts a decimal string into a byte.
(*@KEY@:END_DESCRIPTION*)
FUNCTION_BLOCK DEC_TO_BYTE

(*Group:Default*)

VAR_INPUT
	DEC :	oscat_STRING10;
END_VAR

VAR_OUTPUT
	DEC_TO_BYTE :	BYTE;
END_VAR

VAR
	i :	INT;
	X :	INT;
	stop :	INT;
END_VAR

(*@KEY@: WORKSHEET
NAME: DEC_TO_BYTE
IEC_LANGUAGE: ST
*)
DEC_TO_BYTE := BYTE#0;
stop := LEN(DEC);
FOR I := 1 TO stop DO
	(* read the first character and subtract 48 to get value in decimal 0 = 48 *)
    X := GET_CHAR(DEC,I);
	(* calculate the value of the digit *)
	IF X > 47 AND X < 58 THEN
		DEC_TO_BYTE := INT_TO_BYTE(_BYTE_TO_INT(DEC_TO_BYTE) * 10 + X - 48);
	END_IF;
END_FOR;

(* revision histroy
hm	20. jun. 2008	rev 1.0
	original release

hm	30. sep.2008	rev 1.1
	changed length of input string from 20 to 10
	corrected an error where decoding of characters 8 and 9 would fail

*)
(*@KEY@: END_WORKSHEET *)
END_FUNCTION_BLOCK

(* ---- DEC_TO_DWORD.ST ---- *)
(*@PROPERTIES_EX@
TYPE: POU
LOCALE: 0
IEC_LANGUAGE: ST
PLC_TYPE: independent
PROC_TYPE: independent
GROUP: STRINGS
*)
(*@KEY@:DESCRIPTION*)
version 1.1	30. sep. 2008
programmer 	hugo
tested by		oscat

DEC_TO_DWORD converts a decimal string into a DWORD.
(*@KEY@:END_DESCRIPTION*)
FUNCTION_BLOCK DEC_TO_DWORD

(*Group:Default*)

VAR_INPUT
	DEC :	oscat_STRING20;
END_VAR

VAR_OUTPUT
	DEC_TO_DWORD :	DWORD;
END_VAR

VAR
	i :	INT;
	X :	INT;
	stop :	INT;
END_VAR

(*@KEY@: WORKSHEET
NAME: DEC_TO_DWORD
IEC_LANGUAGE: ST
*)
DEC_TO_DWORD := DWORD#0;
stop := LEN(DEC);
FOR I := 1 TO stop DO
	(* read the first character and subtract 48 to get value in decimal 0 = 48 *)
    X := GET_CHAR(DEC,I);
	(* calculate the value of the digit *)
	IF X > 47 AND X < 58 THEN
		DEC_TO_DWORD := UDINT_TO_DWORD(DWORD_TO_UDINT(DEC_TO_DWORD) * UDINT#10 + _INT_TO_UDINT(X) - UDINT#48);
	END_IF;
END_FOR;

(*
version 1.1	30. sep. 2008
programmer 	hugo
tested by		oscat

DEC_TO_DWORD converts a decimal string into a DWORD.

*)
(*@KEY@: END_WORKSHEET *)
END_FUNCTION_BLOCK

(* ---- DEC_TO_INT.ST ---- *)
(*@PROPERTIES_EX@
TYPE: POU
LOCALE: 0
IEC_LANGUAGE: ST
PLC_TYPE: independent
PROC_TYPE: independent
GROUP: STRINGS
*)
(*@KEY@:DESCRIPTION*)
version 1.1	30. sep. 2008
programmer 	hugo
tested by	oscat

DEC_TO_INT converts a decimal string into an Integer.
(*@KEY@:END_DESCRIPTION*)
FUNCTION_BLOCK DEC_TO_INT

(*Group:Default*)

VAR_INPUT
	DEC :	oscat_STRING10;
END_VAR

VAR_OUTPUT
	DEC_TO_INT :	INT;
END_VAR

VAR
	i :	INT;
	X :	INT;
	sign :	BOOL;
	stop :	INT;
END_VAR

(*@KEY@: WORKSHEET
NAME: DEC_TO_INT
IEC_LANGUAGE: ST
*)
DEC_TO_INT := 0;
sign := FALSE;
stop := LEN(dec);
FOR I := 1 TO stop DO
	(* read the first character and subtract 48 to get value in decimal 0 = 48 *)
    X := GET_CHAR(DEC,I);
	(* calculate the value of the digit *)
	IF X > 47 AND X < 58 THEN
		DEC_TO_INT := DEC_TO_INT * 10 + X - 48;
	ELSIF X = 45 AND DEC_TO_INT = 0 THEN
		sign := TRUE;
	END_IF;
END_FOR;
IF sign THEN DEC_TO_INT := -DEC_TO_INT; END_IF;

(* revision histroy
hm	20. jun. 2008	rev 1.0
	original release

hm	30. sep. 2008	rev 1.1
	changed length of input string from 20 to 10
	corrected an error where decoding of characters 8 and 9 would fail
*)
(*@KEY@: END_WORKSHEET *)
END_FUNCTION_BLOCK

(* ---- DEG_TO_DIR.ST ---- *)
(*@PROPERTIES_EX@
TYPE: POU
LOCALE: 0
IEC_LANGUAGE: ST
PLC_TYPE: independent
PROC_TYPE: independent
GROUP: ENGINEERING.CONVERSION
*)
(*@KEY@:DESCRIPTION*)
version 1.1	22. oct. 2008
programmer 	hugo
tested by	oscat

this function converts degrees in compass direction.
the function supports output in english (L=0) and german (L=1)
(*@KEY@:END_DESCRIPTION*)
FUNCTION_BLOCK DEG_TO_DIR

(*Group:Default*)

VAR_INPUT
	DEG :	INT;
	N :	INT;
	L :	INT;
END_VAR

VAR_OUTPUT
	DEG_TO_DIR :	oscat_STRING3;
END_VAR

VAR
	ly :	INT;
	y :	INT;
	SETUP_DIRS :	SETUP_DIRS;
	DIRS :	oscat_DIRS;
	SETUP_LANGUAGE :	SETUP_LANGUAGE;
	LANGUAGE :	oscat_LANGUAGE;
END_VAR

(*@KEY@: WORKSHEET
NAME: DEG_TO_DIR
IEC_LANGUAGE: ST
*)
SETUP_DIRS(DIRS:=DIRS);
DIRS:=SETUP_DIRS.DIRS;
SETUP_LANGUAGE(LANGUAGE:=LANGUAGE);
LANGUAGE:=SETUP_LANGUAGE.LANGUAGE;

IF L = 0 THEN ly := LANGUAGE.DEFAULT; ELSE ly := MIN(L, LANGUAGE.LMAX); END_IF;
y := ((WORD_TO_INT(SHL(INT_TO_WORD(DEG),N-1)) + 45) / 90) MOD WORD_TO_INT(SHL(WORD#2,N))* WORD_TO_INT(SHR(WORD#8,N));
DEG_TO_DIR := DIRS[ly][y];

(*
DIR := ((SHL(DEG,N-1) + 45) / 90) MOD SHL(INT#2,N);
explanation :
DIR is calculated BY the following formula:
DIR := ((DIR + 45) / 90) MOD 4 if N = 1 digit
North = 0, East = 1 ....
DIR := ((DIR + 22,5) / 45) MOD 8 if N = 2 digit
convert to integer calculation
DIR := ((DIR*2 + 45) / 90) MOD 8
N = 0, NE = 1 ....
ther above formula replaces 2^N with shift for performance
*)

(* revision histroy
hm	11. jun. 2008	rev 1.0
	original release

hm	22. oct. 2008	rev 1.1
	changed size of string variables to 30
*)
(*@KEY@: END_WORKSHEET *)
END_FUNCTION_BLOCK

(* ---- DEL_CHARS.ST ---- *)
(*@PROPERTIES_EX@
TYPE: POU
LOCALE: 0
IEC_LANGUAGE: ST
PLC_TYPE: independent
PROC_TYPE: independent
GROUP: STRINGS
*)
(*@KEY@:DESCRIPTION*)
version 1.0	18. jun. 2008
programmer 	hugo
tested by	oscat

del_chars deletes all characters from a string which are specified in CX.
(*@KEY@:END_DESCRIPTION*)
FUNCTION_BLOCK DEL_CHARS

(*Group:x*)

VAR_INPUT
	IN :	oscat_STRING250;
	CX :	STRING;
END_VAR

VAR_OUTPUT
	DEL_CHARS :	oscat_STRING250;
END_VAR

VAR
	pos :	INT;
	stop :	INT;
	char :	oscat_STRING1;
END_VAR

(*@KEY@: WORKSHEET
NAME: DEL_CHARS
IEC_LANGUAGE: ST
*)
(* copy input string *)
DEL_CHARS := IN;
stop := LEN(in);
pos := 1;
WHILE pos <= stop DO
    char := MID(DEL_CHARS, 1, pos);
	IF FIND(cx,char) > 0 THEN
		(* wrong chracter needs to be deleted *)
		DEL_CHARS := DELETE(DEL_CHARS, 1, pos);
		stop := stop - 1;	(* the string is one character shorter now *)
	ELSE
		(* charcter not found skip to next one *)
		pos := pos + 1;
	END_IF;
END_WHILE;

(* revision history

hm		18. jun. 2008	rev 1.0
	original version
*)

(*@KEY@: END_WORKSHEET *)
END_FUNCTION_BLOCK

(* ---- DELAY.ST ---- *)
(*@PROPERTIES_EX@
TYPE: POU
LOCALE: 0
IEC_LANGUAGE: ST
PLC_TYPE: independent
PROC_TYPE: independent
GROUP: ENGINEERING.SIGNAL_PROCESSING
*)
(*@KEY@:DESCRIPTION*)
version 1.5	23. mar. 2009
programmer 	hugo
tested by	oscat

this function block delays input values by each programm cycle
after N+1 cycles the in value has shifted to the out.
N can be any alue from 0 .. 32
if n = 0 the input will be present on the output without a delay.
f N > 32 then the output will be delayed by 32 cycles.
any high on rst will load the buffer with in.

(*@KEY@:END_DESCRIPTION*)
FUNCTION_BLOCK DELAY

(*Group:Default*)

VAR_INPUT
	IN :	REAL;
	N :	INT;
	RST :	BOOL;
END_VAR

VAR_OUTPUT
	OUT :	REAL;
END_VAR

VAR
	buf :	oscat_delay_buf;
	i :	INT;
	init :	BOOL;
	stop :	INT;
END_VAR

(*@KEY@: WORKSHEET
NAME: DELAY
IEC_LANGUAGE: ST
*)
stop := LIMIT(0,N,32) - 1;
IF rst OR NOT init THEN
	init := TRUE;
	FOR i := 0 TO stop DO buf[i] := in; END_FOR;
	out := in;
	i := 0;
ELSIF stop < 0 THEN
	out := in;
ELSE
	out := buf[i];
	buf[i] := in;
	i := INC1(i, N);
END_IF;

(* revision history
hm 1.10.2006		rev 1.1
	corrected error in buffer management

hm 19.1.2007		rev 1.2
	changed reset to load the value of in instead of 0

hm	27. oct. 2008	rev 1.3
	improved performance

hm	23. feb.2009	rev 1.4
	corrected an index problem

hm	23. mar. 2009	rev 1.5
	corrected non standard write to input N

*)
(*@KEY@: END_WORKSHEET *)
END_FUNCTION_BLOCK

(* ---- DELAY_4.ST ---- *)
(*@PROPERTIES_EX@
TYPE: POU
LOCALE: 0
IEC_LANGUAGE: ST
PLC_TYPE: independent
PROC_TYPE: independent
GROUP: ENGINEERING.SIGNAL_PROCESSING
*)
(*@KEY@:DESCRIPTION*)
version 1.1	19 jan 2007
programmer 	hugo
tested by	tobias

this function block delays input values by each programm cycle
after 4 cycles the in value has shifted to the out 4 and will be discarded after the next cycle
the blocks can be cascaded.
(*@KEY@:END_DESCRIPTION*)
FUNCTION_BLOCK DELAY_4

(*Group:Default*)

VAR_INPUT
	IN :	REAL;
END_VAR

VAR_OUTPUT
	OUT1 :	REAL;
	OUT2 :	REAL;
	OUT3 :	REAL;
	OUT4 :	REAL;
END_VAR

VAR
	temp :	REAL;
END_VAR

(*@KEY@: WORKSHEET
NAME: DELAY_4
IEC_LANGUAGE: ST
*)
out4 := out3;
out3 := out2;
out2 := out1;
out1 := temp;
temp := in;

(* revision history

hm 19.1.2007	rev 1.1
	added variable temp to add 1 delay  for q1

*)
(*@KEY@: END_WORKSHEET *)
END_FUNCTION_BLOCK

(* ---- DIR_TO_DEG.ST ---- *)
(*@PROPERTIES_EX@
TYPE: POU
LOCALE: 0
IEC_LANGUAGE: ST
PLC_TYPE: independent
PROC_TYPE: independent
GROUP: ENGINEERING.CONVERSION
*)
(*@KEY@:DESCRIPTION*)
version 1.1	22. oct. 2008
programmer 	hugo
tested by	oscat

this function converts compass directions to degrees
it will recognize up to 3 letter directions in english and german writing.
(*@KEY@:END_DESCRIPTION*)
FUNCTION_BLOCK DIR_TO_DEG

(*Group:Default*)

VAR_INPUT
	DIR :	oscat_STRING3;
	L :	INT;
END_VAR

VAR_OUTPUT
	DIR_TO_DEG :	INT;
END_VAR

VAR
	ly :	INT;
	i :	INT;
	SETUP_DIRS :	SETUP_DIRS;
	DIRS :	oscat_DIRS;
	SETUP_LANGUAGE :	SETUP_LANGUAGE;
	LANGUAGE :	oscat_LANGUAGE;
END_VAR

(*@KEY@: WORKSHEET
NAME: DIR_TO_DEG
IEC_LANGUAGE: ST
*)
SETUP_DIRS(DIRS:=DIRS);
DIRS:=SETUP_DIRS.DIRS;
SETUP_LANGUAGE(LANGUAGE:=LANGUAGE);
LANGUAGE:=SETUP_LANGUAGE.LANGUAGE;

IF L = 0 THEN ly := LANGUAGE.DEFAULT; ELSE ly := MIN(L, LANGUAGE.LMAX); END_IF;
FOR i := 0 TO 15 DO
	IF EQ_STRING(DIRS[ly][i],DIR) THEN EXIT; END_IF;
END_FOR;
DIR_TO_DEG := WORD_TO_INT(SHR_WORD(INT_TO_WORD(i * 45 + 1), 1));

(* revision histroy
hm	22. oct. 2008	rev 1.1
	original release

*)
(*@KEY@: END_WORKSHEET *)
END_FUNCTION_BLOCK

(* ---- DRIVER_1.ST ---- *)
(*@PROPERTIES_EX@
TYPE: POU
LOCALE: 0
IEC_LANGUAGE: ST
PLC_TYPE: independent
PROC_TYPE: independent
GROUP: ENGINEERING.AUTOMATION
*)
(*@KEY@:DESCRIPTION*)
version 1.0	2 jan 2008
programmer 	hugo
tested by	tobias

driver_1 is a multi purpose driver.
a rising edge in in sets the output high if toggle is flase. while toggle is true, a rising edge on in toggles the output Q.
if a timeout is specified the output q will be reset to false automatically after the timeout has elapsed.
a asynchronous reset and set will force the output high or low respectively.
(*@KEY@:END_DESCRIPTION*)
FUNCTION_BLOCK DRIVER_1

(*Group:Default*)

VAR_INPUT
	SET :	BOOL;
	IN :	BOOL;
	RST :	BOOL;
	TOGGLE_MODE :	BOOL;
	TIMEOUT :	TIME;
END_VAR

VAR_OUTPUT
	Q :	BOOL;
END_VAR

VAR
	off :	TON;
	edge :	BOOL;
END_VAR

(*@KEY@: WORKSHEET
NAME: DRIVER_1
IEC_LANGUAGE: ST
*)
IF off.Q THEN Q := FALSE; END_IF;
IF rst THEN
	Q := FALSE;
ELSIF set THEN
	Q := TRUE;
ELSIF IN AND NOT edge THEN
	IF toggle_mode THEN q := NOT Q; ELSE q := TRUE; END_IF;
END_IF;
edge := in;
IF timeout > t#0s THEN off(in := Q, PT := Timeout); END_IF;

(* revision history
hm	2. jan 2008		rev 1.0
	original version

*)
(*@KEY@: END_WORKSHEET *)
END_FUNCTION_BLOCK

(* ---- DRIVER_4.ST ---- *)
(*@PROPERTIES_EX@
TYPE: POU
LOCALE: 0
IEC_LANGUAGE: ST
PLC_TYPE: independent
PROC_TYPE: independent
GROUP: ENGINEERING.AUTOMATION
*)
(*@KEY@:DESCRIPTION*)
version 1.0	2 jan 2008
programmer 	hugo
tested by	tobias

driver_4 is a multi purpose driver.
a rising edge in in sets the output high if toggle is flase. while toggle is true, a rising edge on in toggles the output Q.
if a timeout is specified the output q will be reset to false automatically after the timeout has elapsed.
a asynchronous reset and set will force the output high or low respectively.
(*@KEY@:END_DESCRIPTION*)
FUNCTION_BLOCK DRIVER_4

(*Group:Default*)

VAR_INPUT
	SET :	BOOL;
	IN0 :	BOOL;
	IN1 :	BOOL;
	IN2 :	BOOL;
	IN3 :	BOOL;
	RST :	BOOL;
	TOGGLE_MODE :	BOOL;
	TIMEOUT :	TIME;
END_VAR

VAR_OUTPUT
	Q0 :	BOOL;
	Q1 :	BOOL;
	Q2 :	BOOL;
	Q3 :	BOOL;
END_VAR

VAR
	d0 :	DRIVER_1;
	d1 :	DRIVER_1;
	d2 :	DRIVER_1;
	d3 :	DRIVER_1;
END_VAR

(*@KEY@: WORKSHEET
NAME: DRIVER_4
IEC_LANGUAGE: ST
*)
D0(Set:=set, in:=in0, rst:=rst, toggle_mode:=toggle_mode, timeout:=timeout);
D1(Set:=set, in:=in1, rst:=rst, toggle_mode:=toggle_mode, timeout:=timeout);
D2(Set:=set, in:=in2, rst:=rst, toggle_mode:=toggle_mode, timeout:=timeout);
D3(Set:=set, in:=in3, rst:=rst, toggle_mode:=toggle_mode, timeout:=timeout);
Q0 := D0.Q;
Q1 := D1.Q;
Q2 := D2.Q;
Q3 := D3.Q;

(* revision history
hm	2. jan 2008		rev 1.0
	original version

*)
(*@KEY@: END_WORKSHEET *)
END_FUNCTION_BLOCK

(* ---- DRIVER_4C.ST ---- *)
(*@PROPERTIES_EX@
TYPE: POU
LOCALE: 0
IEC_LANGUAGE: ST
PLC_TYPE: independent
PROC_TYPE: independent
GROUP: ENGINEERING.AUTOMATION
*)
(*@KEY@:DESCRIPTION*)
version 1.0	23. mar. 2009
programmer 	hugo
tested by	tobias

driver_4C is a multi purpose driver.
a rising edge on in switches from S0 state S1 and the next edge to state S2 and so on.
in state S0 all outputs Q are FALSE.
The stet of the Outputs in any state S? is configurable with setup variables.
The variables S1..S5 define the states, while the sequence is terminated when a state Variable S? = 0.
The lower bits 0..3 of the state vars S? are corresponding to the Outputs Q0..Q3

(*@KEY@:END_DESCRIPTION*)
FUNCTION_BLOCK DRIVER_4C

(*Group:Default*)

VAR_INPUT
	IN :	BOOL;
	RST :	BOOL;
	TIMEOUT :	TIME;
	SX :	oscat_DRIVER_4C;
END_VAR

VAR_OUTPUT
	SN :	INT;
	Q0 :	BOOL;
	Q1 :	BOOL;
	Q2 :	BOOL;
	Q3 :	BOOL;
END_VAR

VAR
	off :	TON;
	edge :	BOOL;
END_VAR

(*@KEY@: WORKSHEET
NAME: DRIVER_4C
IEC_LANGUAGE: ST
*)
IF RST OR off.Q THEN
	SN := 0;
ELSIF IN AND NOT edge THEN
	SN := SN + 1;
	IF SN > 7 OR SX[SN] = BYTE#0 THEN SN := 0; END_IF;
END_IF;
edge := in;
IF SN > 0 THEN
	Q0 := (SX[SN] AND BYTE#1) > BYTE#0;
	Q1 := (SX[SN] AND BYTE#2) > BYTE#0;
	Q2 := (SX[SN] AND BYTE#4) > BYTE#0;
	Q3 := (SX[SN] AND BYTE#8) > BYTE#0;
ELSE
	Q0 := FALSE;
	Q1 := FALSE;
	Q2 := FALSE;
	Q3 := FALSE;
END_IF;

(* maximaum timeout *)
IF timeout > t#0s THEN off(in := SN > 0, PT := Timeout); END_IF;

(* revision history
hm	23. mar. 2009	rev 1.0
	original version

*)
(*@KEY@: END_WORKSHEET *)
END_FUNCTION_BLOCK

(* ---- DT2_TO_SDT.ST ---- *)
(*@PROPERTIES_EX@
TYPE: POU
LOCALE: 0
IEC_LANGUAGE: ST
PLC_TYPE: independent
PROC_TYPE: independent
GROUP: TIME_DATE
*)
(*@KEY@:DESCRIPTION*)
version 1.0	18. oct 2008
programmer 	hugo
tested by	oscat

converts date and time of day to Structured date time (SDT)
(*@KEY@:END_DESCRIPTION*)
FUNCTION_BLOCK DT2_TO_SDT

(*Group:Default*)

VAR_INPUT
	DI :	UDINT;
	TI :	UDINT;
END_VAR

VAR_OUTPUT
	SDT :	oscat_SDT;
END_VAR

(*@KEY@: WORKSHEET
NAME: DT2_TO_SDT
IEC_LANGUAGE: ST
*)
SDT.YEAR := YEAR_OF_DATE(di);
SDT.MONTH := MONTH_OF_DATE(di);
SDT.DAY := DAY_OF_MONTH(di);
SDT.WEEKDAY := DAY_OF_WEEK(di);
SDT.MS := UDINT_TO_INT(ti MOD UDINT#1000);
SDT.SECOND := UDINT_TO_INT((ti / UDINT#1000) MOD UDINT#60);
SDT.MINUTE := UDINT_TO_INT((ti / UDINT#60000) MOD UDINT#60);
SDT.HOUR := UDINT_TO_INT(ti / UDINT#3600000);

(* revision history

hm 18. oct. 2008	rev 1.0
	original version

*)
(*@KEY@: END_WORKSHEET *)
END_FUNCTION_BLOCK

(* ---- DT_SIMU.ST ---- *)
(*@PROPERTIES_EX@
TYPE: POU
LOCALE: 0
IEC_LANGUAGE: ST
PLC_TYPE: independent
PROC_TYPE: independent
GROUP: ENGINEERING.MEASUREMENTS
*)
(*@KEY@:DESCRIPTION*)
version 1.2	8. mar. 2009
programmer 	hugo
tested by	oscat

DT_SIMU simulates a real time clock and can be adjusted to different speeds
it can also be used in simulation to simulate a real time clock.
the peed of the clock can be increased or decreased to debug timers.
with the input start a start date-time can be specified.
(*@KEY@:END_DESCRIPTION*)
FUNCTION_BLOCK DT_SIMU

(*Group:Default*)

VAR_INPUT
	START :	UDINT;
	SPEED :	REAL := 1.0;
END_VAR

VAR_OUTPUT
	DTS :	UDINT;
END_VAR

VAR
	tc :	UDINT;
	init :	BOOL;
	last :	UDINT;
	tx :	UDINT;
	td :	UDINT;
	T_PLC_MS :	T_PLC_MS;
END_VAR

(*@KEY@: WORKSHEET
NAME: DT_SIMU
IEC_LANGUAGE: ST
*)
(* read system timer *)
T_PLC_MS();
tx:= T_PLC_MS.T_PLC_MS;
tc := _REAL_TO_UDINT(UDINT_TO_REAL(tx - last) * speed);

IF NOT init THEN
	init := TRUE;
	DTS := Start;
	tc := UDINT#0;
	last := tx;
ELSIF SPEED = 0.0 THEN
	DTS := DTS + UDINT#1;
ELSIF tc >= UDINT#1000 THEN
	td := (tc / UDINT#1000) * UDINT#1000;
	DTS := DTS + td;
	last := last + _REAL_TO_UDINT(UDINT_TO_REAL(td) / speed);
END_IF;

(* revision history
hm	11. sep. 2008	rev 1.0
	original version

hm	16. nov	2008	rev 1.1
	added type conversions for compatibility reasons

hm	8.	mar. 2009	rev 1.2
	added increment by cycle mode
*)
(*@KEY@: END_WORKSHEET *)
END_FUNCTION_BLOCK

(* ---- DT_TO_SDT.ST ---- *)
(*@PROPERTIES_EX@
TYPE: POU
LOCALE: 0
IEC_LANGUAGE: ST
PLC_TYPE: independent
PROC_TYPE: independent
GROUP: TIME_DATE
*)
(*@KEY@:DESCRIPTION*)
version 1.0	18. oct 2008
programmer 	hugo
tested by	oscat

converts date_time to Structured date time (SDT)
(*@KEY@:END_DESCRIPTION*)
FUNCTION_BLOCK DT_TO_SDT

(*Group:Default*)

VAR_INPUT
	DTI :	UDINT;
END_VAR

VAR_OUTPUT
	SDT :	oscat_SDT;
END_VAR

VAR
	tmp :	UDINT;
	tdt :	UDINT;
END_VAR

(*@KEY@: WORKSHEET
NAME: DT_TO_SDT
IEC_LANGUAGE: ST
*)
tmp := DT_TO_DATE(dti);
tdt := dti - tmp;
SDT.YEAR := YEAR_OF_DATE(tmp);
SDT.MONTH := MONTH_OF_DATE(tmp);
SDT.DAY := DAY_OF_MONTH(tmp);
SDT.WEEKDAY := DAY_OF_WEEK(tmp);
SDT.SECOND := UDINT_TO_INT(tdt MOD UDINT#60);
SDT.MINUTE := UDINT_TO_INT((tdt / UDINT#60) MOD UDINT#60);
SDT.HOUR := UDINT_TO_INT(tdt / UDINT#3600);

(* revision history

hm 18. oct. 2008	rev 1.0
	original version

*)
(*@KEY@: END_WORKSHEET *)
END_FUNCTION_BLOCK
